LIN {X 0,Y 309.609,Z 476.03,A -85,B 0,C 180,E1 14397.201,E2 14397.201} C_VEL
LIN {X 0,Y 309.614,Z 476.03,A -85,B 0,C 180,E1 14402.807,E2 14402.807} C_VEL
LIN {X 0,Y 308.871,Z 476.03,A -85,B 0,C 180,E1 14411.359,E2 14411.359} C_VEL
LIN {X 0,Y 308.57,Z 476.03,A -85,B 0,C 180,E1 14417.126,E2 14417.126} C_VEL
LIN {X 0,Y 308.226,Z 476.03,A -85,B 0,C 180,E1 14423.143,E2 14423.143} C_VEL
LIN {X 0,Y 307.931,Z 476.03,A -85,B 0,C 180,E1 14429.455,E2 14429.455} C_VEL
LIN {X 0,Y 307.612,Z 476.03,A -85,B 0,C 180,E1 14438.044,E2 14438.044} C_VEL
LIN {X 0,Y 307.589,Z 476.399,A -85,B 0,C 180,E1 14444.592,E2 14444.592} C_VEL
LIN {X 0,Y 310.21,Z 481.903,A -85,B 0,C 180,E1 14445.728,E2 14445.728} C_VEL
LIN {X 0,Y 323.143,Z 502.52,A -85,B 0,C 180,E1 14450.241,E2 14450.241} C_VEL
LIN {X 0,Y 336.192,Z 527.008,A -85,B 0,C 180,E1 14454.493,E2 14454.493} C_VEL
LIN {X 0,Y 347.113,Z 555.503,A -85,B 0,C 180,E1 14458.945,E2 14458.945} C_VEL
LIN {X 0,Y 352.766,Z 578.755,A -85,B 0,C 180,E1 14462.454,E2 14462.454} C_VEL
LIN {X 0,Y 343.722,Z 612.822,A -85,B 0,C 180,E1 14466.127,E2 14466.127} C_VEL
LIN {X 0,Y 334.039,Z 643.34,A -85,B 0,C 180,E1 14470.815,E2 14470.815} C_VEL
LIN {X 0,Y 325.306,Z 668.498,A -85,B 0,C 180,E1 14476.2,E2 14476.2} C_VEL
LIN {X 0,Y 318.194,Z 689.408,A -85,B 0,C 180,E1 14482.481,E2 14482.481} C_VEL
LIN {X 0,Y 313.479,Z 704.958,A -85,B 0,C 180,E1 14489.309,E2 14489.309} C_VEL
LIN {X 0,Y 311.322,Z 714.339,A -85,B 0,C 180,E1 14495.582,E2 14495.582} C_VEL
LIN {X 0,Y 309.931,Z 719.848,A -85,B 0,C 180,E1 14502.293,E2 14502.293} C_VEL
LIN {X 0,Y 309.637,Z 721.106,A -85,B 0,C 180,E1 14507.062,E2 14507.062} C_VEL
LIN {X 0,Y 310.382,Z 718.696,A -85,B 0,C 180,E1 14514.46,E2 14514.46} C_VEL
LIN {X 0,Y 312.319,Z 711.622,A -85,B 0,C 180,E1 14521.411,E2 14521.411} C_VEL
LIN {X 0,Y 316.175,Z 699.192,A -85,B 0,C 180,E1 14528.503,E2 14528.503} C_VEL
LIN {X 0,Y 322.949,Z 681.144,A -85,B 0,C 180,E1 14535.309,E2 14535.309} C_VEL
LIN {X 0,Y 332.145,Z 658.16,A -85,B 0,C 180,E1 14541.336,E2 14541.336} C_VEL
LIN {X 0,Y 342.684,Z 630.258,A -85,B 0,C 180,E1 14546.482,E2 14546.482} C_VEL
LIN {X 0,Y 352.98,Z 599.194,A -85,B 0,C 180,E1 14550.557,E2 14550.557} C_VEL
LIN {X 0,Y 356.508,Z 587.102,A -85,B 0,C 180,E1 14551.803,E2 14551.803} C_VEL
LIN {X 0,Y 356.262,Z 585.186,A -85,B 0,C 180,E1 14552.126,E2 14552.126} C_VEL
LIN {X 0,Y 336.094,Z 594.919,A -85,B 0,C 180,E1 14554.892,E2 14554.892} C_VEL
LIN {X 0,Y 320.136,Z 599.709,A -85,B 0,C 180,E1 14558.13,E2 14558.13} C_VEL
LIN {X 0,Y 319.686,Z 600.582,A -85,B 0,C 180,E1 14558.463,E2 14558.463} C_VEL
LIN {X 0,Y 316.983,Z 624.334,A -85,B 0,C 180,E1 14562.389,E2 14562.389} C_VEL
LIN {X 0,Y 314.808,Z 644.294,A -85,B 0,C 180,E1 14567.144,E2 14567.144} C_VEL
LIN {X 0,Y 313.633,Z 658.734,A -85,B 0,C 180,E1 14572.387,E2 14572.387} C_VEL
LIN {X 0,Y 313.388,Z 666.672,A -85,B 0,C 180,E1 14577.227,E2 14577.227} C_VEL
LIN {X 0,Y 313.677,Z 669.126,A -85,B 0,C 180,E1 14579.996,E2 14579.996} C_VEL
LIN {X 0,Y 314.606,Z 669.657,A -85,B 0,C 180,E1 14585.519,E2 14585.519} C_VEL
LIN {X 0,Y 316.918,Z 664.101,A -85,B 0,C 180,E1 14591.012,E2 14591.012} C_VEL
LIN {X 0,Y 320.125,Z 653.696,A -85,B 0,C 180,E1 14595.776,E2 14595.776} C_VEL
LIN {X 0,Y 324.288,Z 637.409,A -85,B 0,C 180,E1 14600.34,E2 14600.34} C_VEL
LIN {X 0,Y 328.84,Z 615.987,A -85,B 0,C 180,E1 14604.294,E2 14604.294} C_VEL
LIN {X 0,Y 333.119,Z 589.74,A -85,B 0,C 180,E1 14607.559,E2 14607.559} C_VEL
LIN {X 0,Y 336.661,Z 558.53,A -85,B 0,C 180,E1 14610.116,E2 14610.116} C_VEL
LIN {X 0,Y 338.184,Z 535.72,A -85,B 0,C 180,E1 14611.463,E2 14611.463} C_VEL
LIN {X 0,Y 341.71,Z 532.148,A -85,B 0,C 180,E1 14612.114,E2 14612.114} C_VEL
LIN {X 0,Y 344.501,Z 534.122,A -85,B 0,C 180,E1 14613.117,E2 14613.117} C_VEL
LIN {X 0,Y 356.019,Z 559.364,A -85,B 0,C 180,E1 14618.453,E2 14618.453} C_VEL
LIN {X 0,Y 362.184,Z 578.437,A -85,B 0,C 180,E1 14621.558,E2 14621.558} C_VEL
LIN {X 0,Y 351.358,Z 622.491,A -85,B 0,C 180,E1 14624.831,E2 14624.831} C_VEL
LIN {X 0,Y 341.461,Z 657.119,A -85,B 0,C 180,E1 14628.505,E2 14628.505} C_VEL
LIN {X 0,Y 331.204,Z 689.072,A -85,B 0,C 180,E1 14633.283,E2 14633.283} C_VEL
LIN {X 0,Y 322.511,Z 716.02,A -85,B 0,C 180,E1 14638.907,E2 14638.907} C_VEL
LIN {X 0,Y 316.055,Z 737.747,A -85,B 0,C 180,E1 14645.179,E2 14645.179} C_VEL
LIN {X 0,Y 312.202,Z 753.977,A -85,B 0,C 180,E1 14651.794,E2 14651.794} C_VEL
LIN {X 0,Y 310.523,Z 765.226,A -85,B 0,C 180,E1 14658.752,E2 14658.752} C_VEL
LIN {X 0,Y 310.158,Z 770.4,A -85,B 0,C 180,E1 14664.396,E2 14664.396} C_VEL
LIN {X 0,Y 310.336,Z 772.13,A -85,B 0,C 180,E1 14670,E2 14670} C_VEL
LIN {X 0,Y 310.165,Z 770.387,A -85,B 0,C 180,E1 14675.602,E2 14675.602} C_VEL
LIN {X 0,Y 310.766,Z 763.954,A -85,B 0,C 180,E1 14682.17,E2 14682.17} C_VEL
LIN {X 0,Y 312.508,Z 751.967,A -85,B 0,C 180,E1 14688.996,E2 14688.996} C_VEL
LIN {X 0,Y 316.833,Z 733.579,A -85,B 0,C 180,E1 14695.853,E2 14695.853} C_VEL
LIN {X 0,Y 323.626,Z 709.884,A -85,B 0,C 180,E1 14702.054,E2 14702.054} C_VEL
LIN {X 0,Y 325.491,Z 703.783,A -85,B 0,C 180,E1 14703.347,E2 14703.347} C_VEL
LIN {X 0,Y 325.165,Z 692.843,A -85,B 0,C 180,E1 14705.761,E2 14705.761} C_VEL
LIN {X 0,Y 325.168,Z 681.265,A -85,B 0,C 180,E1 14708.078,E2 14708.078} C_VEL
LIN {X 0,Y 334.706,Z 649.033,A -85,B 0,C 180,E1 14712.51,E2 14712.51} C_VEL
LIN {X 0,Y 344.112,Z 612.413,A -85,B 0,C 180,E1 14716.096,E2 14716.096} C_VEL
LIN {X 0,Y 351.392,Z 578.99,A -85,B 0,C 180,E1 14718.568,E2 14718.568} C_VEL
LIN {X 0,Y 336.934,Z 544.114,A -85,B 0,C 180,E1 14723.905,E2 14723.905} C_VEL
LIN {X 0,Y 320.974,Z 511.874,A -85,B 0,C 180,E1 14729.732,E2 14729.732} C_VEL
LIN {X 0,Y 306.924,Z 488.255,A -85,B 0,C 180,E1 14735.215,E2 14735.215} C_VEL
LIN {X 0,Y 302.442,Z 481.461,A -85,B 0,C 180,E1 14737.135,E2 14737.135} C_VEL
LIN {X 0,Y 300.284,Z 476.03,A -85,B 0,C 180,E1 14738.37,E2 14738.37} C_VEL
LIN {X 0,Y 300.741,Z 476.03,A -85,B 0,C 180,E1 14745.426,E2 14745.426} C_VEL
LIN {X 0,Y 301.409,Z 476.03,A -85,B 0,C 180,E1 14754.239,E2 14754.239} C_VEL
LIN {X 0,Y 301.9,Z 476.03,A -85,B 0,C 180,E1 14760.004,E2 14760.004} C_VEL
LIN {X 0,Y 301.407,Z 476.03,A -85,B 0,C 180,E1 14765.77,E2 14765.77} C_VEL
LIN {X 0,Y 300.719,Z 476.03,A -85,B 0,C 180,E1 14774.585,E2 14774.585} C_VEL
LIN {X 0,Y 300.42,Z 476.03,A -85,B 0,C 180,E1 14780.662,E2 14780.662} C_VEL
LIN {X 0,Y 300.101,Z 476.03,A -85,B 0,C 180,E1 14787.009,E2 14787.009} C_VEL
LIN {X 0,Y 299.748,Z 476.03,A -85,B 0,C 180,E1 14793.757,E2 14793.757} C_VEL
LIN {X 0,Y 299.724,Z 476.285,A -85,B 0,C 180,E1 14802.203,E2 14802.203} C_VEL
LIN {X 0,Y 302.277,Z 481.846,A -85,B 0,C 180,E1 14803.462,E2 14803.462} C_VEL
LIN {X 0,Y 316.05,Z 503.587,A -85,B 0,C 180,E1 14808.7,E2 14808.7} C_VEL
LIN {X 0,Y 328.607,Z 526.591,A -85,B 0,C 180,E1 14813.002,E2 14813.002} C_VEL
LIN {X 0,Y 339.745,Z 555.047,A -85,B 0,C 180,E1 14817.67,E2 14817.67} C_VEL
LIN {X 0,Y 346.253,Z 581.175,A -85,B 0,C 180,E1 14821.795,E2 14821.795} C_VEL
LIN {X 0,Y 336.754,Z 615.416,A -85,B 0,C 180,E1 14825.601,E2 14825.601} C_VEL
LIN {X 0,Y 327.378,Z 643.814,A -85,B 0,C 180,E1 14830.057,E2 14830.057} C_VEL
LIN {X 0,Y 318.262,Z 669.058,A -85,B 0,C 180,E1 14835.537,E2 14835.537} C_VEL
LIN {X 0,Y 311.113,Z 689.02,A -85,B 0,C 180,E1 14841.605,E2 14841.605} C_VEL
LIN {X 0,Y 306,Z 704.987,A -85,B 0,C 180,E1 14848.583,E2 14848.583} C_VEL
LIN {X 0,Y 303.42,Z 715.365,A -85,B 0,C 180,E1 14855.728,E2 14855.728} C_VEL
LIN {X 0,Y 302.19,Z 720.102,A -85,B 0,C 180,E1 14861.562,E2 14861.562} C_VEL
LIN {X 0,Y 301.746,Z 721.759,A -85,B 0,C 180,E1 14867.561,E2 14867.561} C_VEL
LIN {X 0,Y 302.329,Z 719.996,A -85,B 0,C 180,E1 14873.62,E2 14873.62} C_VEL
LIN {X 0,Y 303.926,Z 714.692,A -85,B 0,C 180,E1 14879.881,E2 14879.881} C_VEL
LIN {X 0,Y 307.433,Z 703.637,A -85,B 0,C 180,E1 14887.234,E2 14887.234} C_VEL
LIN {X 0,Y 313.533,Z 688.033,A -85,B 0,C 180,E1 14893.962,E2 14893.962} C_VEL
LIN {X 0,Y 322.849,Z 665.785,A -85,B 0,C 180,E1 14900.564,E2 14900.564} C_VEL
LIN {X 0,Y 333.538,Z 639.537,A -85,B 0,C 180,E1 14905.973,E2 14905.973} C_VEL
LIN {X 0,Y 344.606,Z 608.868,A -85,B 0,C 180,E1 14910.476,E2 14910.476} C_VEL
LIN {X 0,Y 349.077,Z 594.477,A -85,B 0,C 180,E1 14912.099,E2 14912.099} C_VEL
LIN {X 0,Y 330.37,Z 602.428,A -85,B 0,C 180,E1 14914.84,E2 14914.84} C_VEL
LIN {X 0,Y 312.096,Z 607.854,A -85,B 0,C 180,E1 14918.66,E2 14918.66} C_VEL
LIN {X 0,Y 311.303,Z 607.869,A -85,B 0,C 180,E1 14919.07,E2 14919.07} C_VEL
LIN {X 0,Y 308.724,Z 630.581,A -85,B 0,C 180,E1 14923.25,E2 14923.25} C_VEL
LIN {X 0,Y 306.627,Z 649.378,A -85,B 0,C 180,E1 14928.244,E2 14928.244} C_VEL
LIN {X 0,Y 305.671,Z 662.626,A -85,B 0,C 180,E1 14933.703,E2 14933.703} C_VEL
LIN {X 0,Y 305.672,Z 669.315,A -85,B 0,C 180,E1 14938.577,E2 14938.577} C_VEL
LIN {X 0,Y 306.155,Z 671.615,A -85,B 0,C 180,E1 14942.83,E2 14942.83} C_VEL
LIN {X 0,Y 308.063,Z 669.42,A -85,B 0,C 180,E1 14948.474,E2 14948.474} C_VEL
LIN {X 0,Y 310.599,Z 662.704,A -85,B 0,C 180,E1 14953.214,E2 14953.214} C_VEL
LIN {X 0,Y 314.735,Z 649.762,A -85,B 0,C 180,E1 14958.216,E2 14958.216} C_VEL
LIN {X 0,Y 319.414,Z 631.57,A -85,B 0,C 180,E1 14962.647,E2 14962.647} C_VEL
LIN {X 0,Y 324.414,Z 607.766,A -85,B 0,C 180,E1 14966.5,E2 14966.5} C_VEL
LIN {X 0,Y 329.026,Z 578.611,A -85,B 0,C 180,E1 14969.642,E2 14969.642} C_VEL
LIN {X 0,Y 332.117,Z 551.912,A -85,B 0,C 180,E1 14971.589,E2 14971.589} C_VEL
LIN {X 0,Y 337.468,Z 544.738,A -85,B 0,C 180,E1 14972.309,E2 14972.309} C_VEL
LIN {X 0,Y 340.537,Z 540.572,A -85,B 0,C 180,E1 14972.717,E2 14972.717} C_VEL
LIN {X 0,Y 351.596,Z 566.201,A -85,B 0,C 180,E1 14978.236,E2 14978.236} C_VEL
LIN {X 0,Y 356.147,Z 581.6,A -85,B 0,C 180,E1 14980.796,E2 14980.796} C_VEL
LIN {X 0,Y 345.155,Z 624.579,A -85,B 0,C 180,E1 14984.082,E2 14984.082} C_VEL
LIN {X 0,Y 334.669,Z 659.139,A -85,B 0,C 180,E1 14987.876,E2 14987.876} C_VEL
LIN {X 0,Y 324.287,Z 689.876,A -85,B 0,C 180,E1 14992.628,E2 14992.628} C_VEL
LIN {X 0,Y 315.042,Z 716.939,A -85,B 0,C 180,E1 14998.486,E2 14998.486} C_VEL
LIN {X 0,Y 308.205,Z 738.6,A -85,B 0,C 180,E1 15005.039,E2 15005.039} C_VEL
LIN {X 0,Y 304.369,Z 754.041,A -85,B 0,C 180,E1 15011.651,E2 15011.651} C_VEL
LIN {X 0,Y 302.674,Z 764.608,A -85,B 0,C 180,E1 15018.457,E2 15018.457} C_VEL
LIN {X 0,Y 302.289,Z 769.775,A -85,B 0,C 180,E1 15024.25,E2 15024.25} C_VEL
LIN {X 0,Y 302.479,Z 771.477,A -85,B 0,C 180,E1 15029.999,E2 15029.999} C_VEL
LIN {X 0,Y 302.296,Z 769.704,A -85,B 0,C 180,E1 15035.749,E2 15035.749} C_VEL
LIN {X 0,Y 302.909,Z 763.208,A -85,B 0,C 180,E1 15042.491,E2 15042.491} C_VEL
LIN {X 0,Y 304.891,Z 750.705,A -85,B 0,C 180,E1 15049.695,E2 15049.695} C_VEL
LIN {X 0,Y 309.48,Z 732.625,A -85,B 0,C 180,E1 15056.515,E2 15056.515} C_VEL
LIN {X 0,Y 316.823,Z 708.164,A -85,B 0,C 180,E1 15062.982,E2 15062.982} C_VEL
LIN {X 0,Y 325.168,Z 681.265,A -85,B 0,C 180,E1 15068.078,E2 15068.078} C_VEL
LIN {X 0,Y 325.431,Z 669.165,A -85,B 0,C 180,E1 15070.295,E2 15070.295} C_VEL
LIN {X 0,Y 325.964,Z 656.299,A -85,B 0,C 180,E1 15072.402,E2 15072.402} C_VEL
LIN {X 0,Y 335.65,Z 620.882,A -85,B 0,C 180,E1 15076.199,E2 15076.199} C_VEL
LIN {X 0,Y 344.722,Z 581.453,A -85,B 0,C 180,E1 15079.278,E2 15079.278} C_VEL
LIN {X 0,Y 330.067,Z 545.357,A -85,B 0,C 180,E1 15085.046,E2 15085.046} C_VEL
LIN {X 0,Y 313.615,Z 512.289,A -85,B 0,C 180,E1 15091.422,E2 15091.422} C_VEL
LIN {X 0,Y 299.519,Z 488.628,A -85,B 0,C 180,E1 15097.433,E2 15097.433} C_VEL
LIN {X 0,Y 295.081,Z 481.89,A -85,B 0,C 180,E1 15099.546,E2 15099.546} C_VEL
LIN {X 0,Y 292.539,Z 476.847,A -85,B 0,C 180,E1 15100.936,E2 15100.936} C_VEL
LIN {X 0,Y 293.021,Z 476.03,A -85,B 0,C 180,E1 15108.077,E2 15108.077} C_VEL
LIN {X 0,Y 293.78,Z 476.03,A -85,B 0,C 180,E1 15117.05,E2 15117.05} C_VEL
LIN {X 0,Y 293.784,Z 476.03,A -85,B 0,C 180,E1 15122.959,E2 15122.959} C_VEL
LIN {X 0,Y 293.006,Z 476.03,A -85,B 0,C 180,E1 15131.933,E2 15131.933} C_VEL
LIN {X 0,Y 292.595,Z 476.03,A -85,B 0,C 180,E1 15138.092,E2 15138.092} C_VEL
LIN {X 0,Y 292.254,Z 476.03,A -85,B 0,C 180,E1 15144.489,E2 15144.489} C_VEL
LIN {X 0,Y 291.907,Z 476.03,A -85,B 0,C 180,E1 15151.248,E2 15151.248} C_VEL
LIN {X 0,Y 291.695,Z 476.599,A -85,B 0,C 180,E1 15159.469,E2 15159.469} C_VEL
LIN {X 0,Y 294.432,Z 481.909,A -85,B 0,C 180,E1 15160.944,E2 15160.944} C_VEL
LIN {X 0,Y 296.791,Z 485.38,A -85,B 0,C 180,E1 15162.033,E2 15162.033} C_VEL
LIN {X 0,Y 311.187,Z 508.02,A -85,B 0,C 180,E1 15167.826,E2 15167.826} C_VEL
LIN {X 0,Y 324.016,Z 532.777,A -85,B 0,C 180,E1 15172.6,E2 15172.6} C_VEL
LIN {X 0,Y 334.089,Z 559.936,A -85,B 0,C 180,E1 15177.227,E2 15177.227} C_VEL
LIN {X 0,Y 339.968,Z 582.863,A -85,B 0,C 180,E1 15181.039,E2 15181.039} C_VEL
LIN {X 0,Y 330.175,Z 616.851,A -85,B 0,C 180,E1 15184.901,E2 15184.901} C_VEL
LIN {X 0,Y 320.145,Z 645.971,A -85,B 0,C 180,E1 15189.587,E2 15189.587} C_VEL
LIN {X 0,Y 310.77,Z 670.877,A -85,B 0,C 180,E1 15195.18,E2 15195.18} C_VEL
LIN {X 0,Y 302.749,Z 692.405,A -85,B 0,C 180,E1 15202.095,E2 15202.095} C_VEL
LIN {X 0,Y 297.782,Z 707.44,A -85,B 0,C 180,E1 15209.272,E2 15209.272} C_VEL
LIN {X 0,Y 295.518,Z 716.37,A -85,B 0,C 180,E1 15215.882,E2 15215.882} C_VEL
LIN {X 0,Y 294.221,Z 721.086,A -85,B 0,C 180,E1 15222.1,E2 15222.1} C_VEL
LIN {X 0,Y 293.861,Z 722.38,A -85,B 0,C 180,E1 15228.009,E2 15228.009} C_VEL
LIN {X 0,Y 294.604,Z 720.448,A -85,B 0,C 180,E1 15234.278,E2 15234.278} C_VEL
LIN {X 0,Y 296.845,Z 713.478,A -85,B 0,C 180,E1 15241.937,E2 15241.937} C_VEL
LIN {X 0,Y 301.07,Z 701.705,A -85,B 0,C 180,E1 15249.215,E2 15249.215} C_VEL
LIN {X 0,Y 308.313,Z 684.584,A -85,B 0,C 180,E1 15256.176,E2 15256.176} C_VEL
LIN {X 0,Y 318.22,Z 662.37,A -85,B 0,C 180,E1 15262.418,E2 15262.418} C_VEL
LIN {X 0,Y 329.501,Z 635.565,A -85,B 0,C 180,E1 15267.723,E2 15267.723} C_VEL
LIN {X 0,Y 340.628,Z 605.233,A -85,B 0,C 180,E1 15271.958,E2 15271.958} C_VEL
LIN {X 0,Y 338.109,Z 604.898,A -85,B 0,C 180,E1 15272.565,E2 15272.565} C_VEL
LIN {X 0,Y 322.886,Z 610.379,A -85,B 0,C 180,E1 15275.034,E2 15275.034} C_VEL
LIN {X 0,Y 303.033,Z 615.082,A -85,B 0,C 180,E1 15279.715,E2 15279.715} C_VEL
LIN {X 0,Y 300.125,Z 638.828,A -85,B 0,C 180,E1 15284.74,E2 15284.74} C_VEL
LIN {X 0,Y 298.442,Z 655.134,A -85,B 0,C 180,E1 15289.768,E2 15289.768} C_VEL
LIN {X 0,Y 297.807,Z 665.902,A -85,B 0,C 180,E1 15294.891,E2 15294.891} C_VEL
LIN {X 0,Y 298.135,Z 671.711,A -85,B 0,C 180,E1 15299.996,E2 15299.996} C_VEL
LIN {X 0,Y 299.258,Z 672.874,A -85,B 0,C 180,E1 15305.803,E2 15305.803} C_VEL
LIN {X 0,Y 301.946,Z 667.982,A -85,B 0,C 180,E1 15311.566,E2 15311.566} C_VEL
LIN {X 0,Y 305.614,Z 658.229,A -85,B 0,C 180,E1 15316.546,E2 15316.546} C_VEL
LIN {X 0,Y 310.068,Z 643.917,A -85,B 0,C 180,E1 15321.018,E2 15321.018} C_VEL
LIN {X 0,Y 315.358,Z 623.654,A -85,B 0,C 180,E1 15325.214,E2 15325.214} C_VEL
LIN {X 0,Y 320.604,Z 598.536,A -85,B 0,C 180,E1 15328.733,E2 15328.733} C_VEL
LIN {X 0,Y 325.036,Z 569.44,A -85,B 0,C 180,E1 15331.5,E2 15331.5} C_VEL
LIN {X 0,Y 332.227,Z 559.13,A -85,B 0,C 180,E1 15332.564,E2 15332.564} C_VEL
LIN {X 0,Y 338.121,Z 551.179,A -85,B 0,C 180,E1 15333.261,E2 15333.261} C_VEL
LIN {X 0,Y 346.556,Z 571.323,A -85,B 0,C 180,E1 15337.702,E2 15337.702} C_VEL
LIN {X 0,Y 350.224,Z 584.949,A -85,B 0,C 180,E1 15340.026,E2 15340.026} C_VEL
LIN {X 0,Y 338.701,Z 627.798,A -85,B 0,C 180,E1 15343.411,E2 15343.411} C_VEL
LIN {X 0,Y 327.65,Z 662.04,A -85,B 0,C 180,E1 15347.337,E2 15347.337} C_VEL
LIN {X 0,Y 316.474,Z 693.235,A -85,B 0,C 180,E1 15352.433,E2 15352.433} C_VEL
LIN {X 0,Y 307.059,Z 719.211,A -85,B 0,C 180,E1 15358.404,E2 15358.404} C_VEL
LIN {X 0,Y 300.103,Z 740.344,A -85,B 0,C 180,E1 15365.232,E2 15365.232} C_VEL
LIN {X 0,Y 296.261,Z 755.274,A -85,B 0,C 180,E1 15372.142,E2 15372.142} C_VEL
LIN {X 0,Y 294.639,Z 765.62,A -85,B 0,C 180,E1 15379.638,E2 15379.638} C_VEL
LIN {X 0,Y 294.403,Z 769.151,A -85,B 0,C 180,E1 15384.096,E2 15384.096} C_VEL
LIN {X 0,Y 294.601,Z 770.82,A -85,B 0,C 180,E1 15389.999,E2 15389.999} C_VEL
LIN {X 0,Y 294.414,Z 769.013,A -85,B 0,C 180,E1 15395.903,E2 15395.903} C_VEL
LIN {X 0,Y 295.046,Z 762.407,A -85,B 0,C 180,E1 15402.867,E2 15402.867} C_VEL
LIN {X 0,Y 297.259,Z 749.623,A -85,B 0,C 180,E1 15410.332,E2 15410.332} C_VEL
LIN {X 0,Y 302.5,Z 730.542,A -85,B 0,C 180,E1 15417.567,E2 15417.567} C_VEL
LIN {X 0,Y 309.973,Z 706.75,A -85,B 0,C 180,E1 15423.875,E2 15423.875} C_VEL
LIN {X 0,Y 319.709,Z 676.68,A -85,B 0,C 180,E1 15429.522,E2 15429.522} C_VEL
LIN {X 0,Y 325.964,Z 656.299,A -85,B 0,C 180,E1 15432.402,E2 15432.402} C_VEL
LIN {X 0,Y 326.557,Z 642.972,A -85,B 0,C 180,E1 15434.403,E2 15434.403} C_VEL
LIN {X 0,Y 326.762,Z 630.968,A -85,B 0,C 180,E1 15436.086,E2 15436.086} C_VEL
LIN {X 0,Y 327.217,Z 629.108,A -85,B 0,C 180,E1 15436.279,E2 15436.279} C_VEL
LIN {X 0,Y 338.217,Z 586.314,A -85,B 0,C 180,E1 15439.759,E2 15439.759} C_VEL
LIN {X 0,Y 330.827,Z 564.854,A -85,B 0,C 180,E1 15443.088,E2 15443.088} C_VEL
LIN {X 0,Y 316.237,Z 532.109,A -85,B 0,C 180,E1 15449.03,E2 15449.03} C_VEL
LIN {X 0,Y 302.744,Z 506.704,A -85,B 0,C 180,E1 15454.763,E2 15454.763} C_VEL
LIN {X 0,Y 291.725,Z 488.604,A -85,B 0,C 180,E1 15460.049,E2 15460.049} C_VEL
LIN {X 0,Y 287.735,Z 482.27,A -85,B 0,C 180,E1 15462.218,E2 15462.218} C_VEL
LIN {X 0,Y 284.853,Z 477.159,A -85,B 0,C 180,E1 15463.996,E2 15463.996} C_VEL
LIN {X 0,Y 284.828,Z 476.03,A -85,B 0,C 180,E1 15464.592,E2 15464.592} C_VEL
LIN {X 0,Y 285.249,Z 476.03,A -85,B 0,C 180,E1 15470.843,E2 15470.843} C_VEL
LIN {X 0,Y 285.872,Z 476.03,A -85,B 0,C 180,E1 15476.969,E2 15476.969} C_VEL
LIN {X 0,Y 285.876,Z 476.03,A -85,B 0,C 180,E1 15483.04,E2 15483.04} C_VEL
LIN {X 0,Y 285.039,Z 476.03,A -85,B 0,C 180,E1 15492.272,E2 15492.272} C_VEL
LIN {X 0,Y 284.633,Z 476.03,A -85,B 0,C 180,E1 15498.616,E2 15498.616} C_VEL
LIN {X 0,Y 284.224,Z 476.03,A -85,B 0,C 180,E1 15505.228,E2 15505.228} C_VEL
LIN {X 0,Y 283.914,Z 476.03,A -85,B 0,C 180,E1 15512.232,E2 15512.232} C_VEL
LIN {X 0,Y 283.745,Z 476.662,A -85,B 0,C 180,E1 15516.321,E2 15516.321} C_VEL
LIN {X 0,Y 286.301,Z 481.851,A -85,B 0,C 180,E1 15517.935,E2 15517.935} C_VEL
LIN {X 0,Y 288.695,Z 484.966,A -85,B 0,C 180,E1 15519.171,E2 15519.171} C_VEL
LIN {X 0,Y 296.918,Z 497.495,A -85,B 0,C 180,E1 15523.117,E2 15523.117} C_VEL
LIN {X 0,Y 311.191,Z 521.574,A -85,B 0,C 180,E1 15528.821,E2 15528.821} C_VEL
LIN {X 0,Y 322.531,Z 546.631,A -85,B 0,C 180,E1 15533.62,E2 15533.62} C_VEL
LIN {X 0,Y 331.022,Z 574.59,A -85,B 0,C 180,E1 15538.464,E2 15538.464} C_VEL
LIN {X 0,Y 333.111,Z 586.916,A -85,B 0,C 180,E1 15540.488,E2 15540.488} C_VEL
LIN {X 0,Y 322.86,Z 620.465,A -85,B 0,C 180,E1 15544.478,E2 15544.478} C_VEL
LIN {X 0,Y 312.305,Z 649.755,A -85,B 0,C 180,E1 15549.422,E2 15549.422} C_VEL
LIN {X 0,Y 302.309,Z 675.137,A -85,B 0,C 180,E1 15555.498,E2 15555.498} C_VEL
LIN {X 0,Y 295.014,Z 693.864,A -85,B 0,C 180,E1 15561.887,E2 15561.887} C_VEL
LIN {X 0,Y 289.935,Z 708.672,A -85,B 0,C 180,E1 15569.252,E2 15569.252} C_VEL
LIN {X 0,Y 287.606,Z 717.372,A -85,B 0,C 180,E1 15576.044,E2 15576.044} C_VEL
LIN {X 0,Y 286.332,Z 721.818,A -85,B 0,C 180,E1 15582.212,E2 15582.212} C_VEL
LIN {X 0,Y 285.97,Z 723.003,A -85,B 0,C 180,E1 15588.523,E2 15588.523} C_VEL
LIN {X 0,Y 287.228,Z 719.947,A -85,B 0,C 180,E1 15596.341,E2 15596.341} C_VEL
LIN {X 0,Y 289.963,Z 712.048,A -85,B 0,C 180,E1 15604.014,E2 15604.014} C_VEL
LIN {X 0,Y 295.487,Z 698.518,A -85,B 0,C 180,E1 15611.77,E2 15611.77} C_VEL
LIN {X 0,Y 304.141,Z 679.702,A -85,B 0,C 180,E1 15618.818,E2 15618.818} C_VEL
LIN {X 0,Y 314.888,Z 656.582,A -85,B 0,C 180,E1 15624.83,E2 15624.83} C_VEL
LIN {X 0,Y 327.425,Z 627.238,A -85,B 0,C 180,E1 15630.138,E2 15630.138} C_VEL
LIN {X 0,Y 332.667,Z 613.469,A -85,B 0,C 180,E1 15632.053,E2 15632.053} C_VEL
LIN {X 0,Y 322.212,Z 615.964,A -85,B 0,C 180,E1 15633.958,E2 15633.958} C_VEL
LIN {X 0,Y 298.724,Z 621.958,A -85,B 0,C 180,E1 15639.215,E2 15639.215} C_VEL
LIN {X 0,Y 294.437,Z 622.432,A -85,B 0,C 180,E1 15640.665,E2 15640.665} C_VEL
LIN {X 0,Y 291.833,Z 644.216,A -85,B 0,C 180,E1 15645.729,E2 15645.729} C_VEL
LIN {X 0,Y 290.368,Z 659.482,A -85,B 0,C 180,E1 15650.996,E2 15650.996} C_VEL
LIN {X 0,Y 289.999,Z 670.065,A -85,B 0,C 180,E1 15657.003,E2 15657.003} C_VEL
LIN {X 0,Y 290.37,Z 672.995,A -85,B 0,C 180,E1 15659.995,E2 15659.995} C_VEL
LIN {X 0,Y 291.585,Z 674.478,A -85,B 0,C 180,E1 15665.956,E2 15665.956} C_VEL
LIN {X 0,Y 294.451,Z 669.947,A -85,B 0,C 180,E1 15671.864,E2 15671.864} C_VEL
LIN {X 0,Y 298.408,Z 660.544,A -85,B 0,C 180,E1 15676.957,E2 15676.957} C_VEL
LIN {X 0,Y 303.782,Z 644.865,A -85,B 0,C 180,E1 15682.007,E2 15682.007} C_VEL
LIN {X 0,Y 309.846,Z 623.218,A -85,B 0,C 180,E1 15686.475,E2 15686.475} C_VEL
LIN {X 0,Y 315.564,Z 597.737,A -85,B 0,C 180,E1 15690.005,E2 15690.005} C_VEL
LIN {X 0,Y 318.84,Z 581.686,A -85,B 0,C 180,E1 15691.703,E2 15691.703} C_VEL
LIN {X 0,Y 325.435,Z 574.296,A -85,B 0,C 180,E1 15692.636,E2 15692.636} C_VEL
LIN {X 0,Y 335.517,Z 561.337,A -85,B 0,C 180,E1 15693.782,E2 15693.782} C_VEL
LIN {X 0,Y 343.109,Z 581.621,A -85,B 0,C 180,E1 15698.148,E2 15698.148} C_VEL
LIN {X 0,Y 344.6,Z 587.31,A -85,B 0,C 180,E1 15699.158,E2 15699.158} C_VEL
LIN {X 0,Y 332.771,Z 629.408,A -85,B 0,C 180,E1 15702.562,E2 15702.562} C_VEL
LIN {X 0,Y 321.142,Z 663.568,A -85,B 0,C 180,E1 15706.594,E2 15706.594} C_VEL
LIN {X 0,Y 309.424,Z 694.498,A -85,B 0,C 180,E1 15711.822,E2 15711.822} C_VEL
LIN {X 0,Y 299.602,Z 720.094,A -85,B 0,C 180,E1 15717.95,E2 15717.95} C_VEL
LIN {X 0,Y 292.308,Z 740.975,A -85,B 0,C 180,E1 15725.023,E2 15725.023} C_VEL
LIN {X 0,Y 288.248,Z 755.995,A -85,B 0,C 180,E1 15732.419,E2 15732.419} C_VEL
LIN {X 0,Y 286.796,Z 765.011,A -85,B 0,C 180,E1 15739.351,E2 15739.351} C_VEL
LIN {X 0,Y 286.536,Z 768.535,A -85,B 0,C 180,E1 15743.933,E2 15743.933} C_VEL
LIN {X 0,Y 286.742,Z 770.165,A -85,B 0,C 180,E1 15749.999,E2 15749.999} C_VEL
LIN {X 0,Y 286.545,Z 768.322,A -85,B 0,C 180,E1 15756.066,E2 15756.066} C_VEL
LIN {X 0,Y 287.186,Z 761.639,A -85,B 0,C 180,E1 15763.226,E2 15763.226} C_VEL
LIN {X 0,Y 289.614,Z 748.777,A -85,B 0,C 180,E1 15770.887,E2 15770.887} C_VEL
LIN {X 0,Y 295.027,Z 730.055,A -85,B 0,C 180,E1 15778.141,E2 15778.141} C_VEL
LIN {X 0,Y 303.169,Z 705.604,A -85,B 0,C 180,E1 15784.743,E2 15784.743} C_VEL
LIN {X 0,Y 312.99,Z 676.292,A -85,B 0,C 180,E1 15790.317,E2 15790.317} C_VEL
LIN {X 0,Y 323.394,Z 642.954,A -85,B 0,C 180,E1 15794.821,E2 15794.821} C_VEL
LIN {X 0,Y 327.217,Z 629.108,A -85,B 0,C 180,E1 15796.279,E2 15796.279} C_VEL
LIN {X 0,Y 328.139,Z 614.723,A -85,B 0,C 180,E1 15798.031,E2 15798.031} C_VEL
LIN {X 0,Y 328.953,Z 599.932,A -85,B 0,C 180,E1 15799.669,E2 15799.669} C_VEL
LIN {X 0,Y 331.587,Z 586.783,A -85,B 0,C 180,E1 15800.728,E2 15800.728} C_VEL
LIN {X 0,Y 317.907,Z 551.766,A -85,B 0,C 180,E1 15806.797,E2 15806.797} C_VEL
LIN {X 0,Y 303.981,Z 522.544,A -85,B 0,C 180,E1 15812.891,E2 15812.891} C_VEL
LIN {X 0,Y 291.587,Z 500.707,A -85,B 0,C 180,E1 15818.831,E2 15818.831} C_VEL
LIN {X 0,Y 284.057,Z 488.673,A -85,B 0,C 180,E1 15822.976,E2 15822.976} C_VEL
LIN {X 0,Y 280.379,Z 482.542,A -85,B 0,C 180,E1 15825.343,E2 15825.343} C_VEL
LIN {X 0,Y 277.277,Z 477.708,A -85,B 0,C 180,E1 15827.472,E2 15827.472} C_VEL
LIN {X 0,Y 277.136,Z 476.03,A -85,B 0,C 180,E1 15828.045,E2 15828.045} C_VEL
LIN {X 0,Y 277.943,Z 476.03,A -85,B 0,C 180,E1 15836.882,E2 15836.882} C_VEL
LIN {X 0,Y 277.947,Z 476.03,A -85,B 0,C 180,E1 15843.127,E2 15843.127} C_VEL
LIN {X 0,Y 277.073,Z 476.03,A -85,B 0,C 180,E1 15852.63,E2 15852.63} C_VEL
LIN {X 0,Y 276.497,Z 476.03,A -85,B 0,C 180,E1 15861.421,E2 15861.421} C_VEL
LIN {X 0,Y 276.082,Z 476.03,A -85,B 0,C 180,E1 15869.58,E2 15869.58} C_VEL
LIN {X 0,Y 275.958,Z 476.521,A -85,B 0,C 180,E1 15872.571,E2 15872.571} C_VEL
LIN {X 0,Y 278.26,Z 481.759,A -85,B 0,C 180,E1 15874.42,E2 15874.42} C_VEL
LIN {X 0,Y 280.861,Z 484.837,A -85,B 0,C 180,E1 15875.982,E2 15875.982} C_VEL
LIN {X 0,Y 289.685,Z 498.023,A -85,B 0,C 180,E1 15880.804,E2 15880.804} C_VEL
LIN {X 0,Y 304.465,Z 522.84,A -85,B 0,C 180,E1 15887.274,E2 15887.274} C_VEL
LIN {X 0,Y 315.256,Z 546.247,A -85,B 0,C 180,E1 15892.058,E2 15892.058} C_VEL
LIN {X 0,Y 323.782,Z 573.558,A -85,B 0,C 180,E1 15897.036,E2 15897.036} C_VEL
LIN {X 0,Y 326.953,Z 588.092,A -85,B 0,C 180,E1 15899.626,E2 15899.626} C_VEL
LIN {X 0,Y 316.727,Z 620.742,A -85,B 0,C 180,E1 15903.565,E2 15903.565} C_VEL
LIN {X 0,Y 306.396,Z 648.51,A -85,B 0,C 180,E1 15908.246,E2 15908.246} C_VEL
LIN {X 0,Y 295.828,Z 674.469,A -85,B 0,C 180,E1 15914.413,E2 15914.413} C_VEL
LIN {X 0,Y 287.998,Z 693.581,A -85,B 0,C 180,E1 15920.926,E2 15920.926} C_VEL
LIN {X 0,Y 282.436,Z 708.678,A -85,B 0,C 180,E1 15928.465,E2 15928.465} C_VEL
LIN {X 0,Y 279.697,Z 718.368,A -85,B 0,C 180,E1 15936.216,E2 15936.216} C_VEL
LIN {X 0,Y 278.399,Z 722.653,A -85,B 0,C 180,E1 15942.566,E2 15942.566} C_VEL
LIN {X 0,Y 278.107,Z 723.626,A -85,B 0,C 180,E1 15949.067,E2 15949.067} C_VEL
LIN {X 0,Y 279.557,Z 720.331,A -85,B 0,C 180,E1 15957.123,E2 15957.123} C_VEL
LIN {X 0,Y 282.716,Z 712.051,A -85,B 0,C 180,E1 15965.102,E2 15965.102} C_VEL
LIN {X 0,Y 288.827,Z 698.228,A -85,B 0,C 180,E1 15972.962,E2 15972.962} C_VEL
LIN {X 0,Y 298.233,Z 679.074,A -85,B 0,C 180,E1 15980.133,E2 15980.133} C_VEL
LIN {X 0,Y 310.22,Z 654.487,A -85,B 0,C 180,E1 15986.424,E2 15986.424} C_VEL
LIN {X 0,Y 322.479,Z 626.679,A -85,B 0,C 180,E1 15991.353,E2 15991.353} C_VEL
LIN {X 0,Y 324.961,Z 620.358,A -85,B 0,C 180,E1 15992.287,E2 15992.287} C_VEL
LIN {X 0,Y 297.852,Z 627.4,A -85,B 0,C 180,E1 15997.834,E2 15997.834} C_VEL
LIN {X 0,Y 285.93,Z 629.711,A -85,B 0,C 180,E1 16001.697,E2 16001.697} C_VEL
LIN {X 0,Y 283.539,Z 649.617,A -85,B 0,C 180,E1 16006.878,E2 16006.878} C_VEL
LIN {X 0,Y 282.404,Z 663.433,A -85,B 0,C 180,E1 16012.238,E2 16012.238} C_VEL
LIN {X 0,Y 282.192,Z 671.157,A -85,B 0,C 180,E1 16016.92,E2 16016.92} C_VEL
LIN {X 0,Y 282.571,Z 674.259,A -85,B 0,C 180,E1 16019.995,E2 16019.995} C_VEL
LIN {X 0,Y 283.906,Z 676.095,A -85,B 0,C 180,E1 16026.118,E2 16026.118} C_VEL
LIN {X 0,Y 286.981,Z 671.927,A -85,B 0,C 180,E1 16032.178,E2 16032.178} C_VEL
LIN {X 0,Y 291.212,Z 662.922,A -85,B 0,C 180,E1 16037.389,E2 16037.389} C_VEL
LIN {X 0,Y 296.884,Z 648.017,A -85,B 0,C 180,E1 16042.482,E2 16042.482} C_VEL
LIN {X 0,Y 303.474,Z 627.02,A -85,B 0,C 180,E1 16047.075,E2 16047.075} C_VEL
LIN {X 0,Y 310.112,Z 600.787,A -85,B 0,C 180,E1 16050.9,E2 16050.9} C_VEL
LIN {X 0,Y 311.364,Z 595.307,A -85,B 0,C 180,E1 16051.543,E2 16051.543} C_VEL
LIN {X 0,Y 317.528,Z 589.368,A -85,B 0,C 180,E1 16052.537,E2 16052.537} C_VEL
LIN {X 0,Y 333.101,Z 571.806,A -85,B 0,C 180,E1 16054.483,E2 16054.483} C_VEL
LIN {X 0,Y 338.742,Z 589.606,A -85,B 0,C 180,E1 16058.191,E2 16058.191} C_VEL
LIN {X 0,Y 326.93,Z 631.065,A -85,B 0,C 180,E1 16061.685,E2 16061.685} C_VEL
LIN {X 0,Y 314.461,Z 665.679,A -85,B 0,C 180,E1 16065.901,E2 16065.901} C_VEL
LIN {X 0,Y 302.143,Z 696.414,A -85,B 0,C 180,E1 16071.324,E2 16071.324} C_VEL
LIN {X 0,Y 291.666,Z 722.249,A -85,B 0,C 180,E1 16077.852,E2 16077.852} C_VEL
LIN {X 0,Y 284.534,Z 741.623,A -85,B 0,C 180,E1 16084.804,E2 16084.804} C_VEL
LIN {X 0,Y 280.256,Z 756.666,A -85,B 0,C 180,E1 16092.713,E2 16092.713} C_VEL
LIN {X 0,Y 278.741,Z 765.787,A -85,B 0,C 180,E1 16100.621,E2 16100.621} C_VEL
LIN {X 0,Y 278.619,Z 769.117,A -85,B 0,C 180,E1 16106.884,E2 16106.884} C_VEL
LIN {X 0,Y 278.675,Z 769.027,A -85,B 0,C 180,E1 16113.114,E2 16113.114} C_VEL
LIN {X 0,Y 278.774,Z 765.351,A -85,B 0,C 180,E1 16119.377,E2 16119.377} C_VEL
LIN {X 0,Y 279.997,Z 756.834,A -85,B 0,C 180,E1 16126.493,E2 16126.493} C_VEL
LIN {X 0,Y 283.899,Z 741.314,A -85,B 0,C 180,E1 16134.414,E2 16134.414} C_VEL
LIN {X 0,Y 290.444,Z 720.953,A -85,B 0,C 180,E1 16141.42,E2 16141.42} C_VEL
LIN {X 0,Y 299.976,Z 694.051,A -85,B 0,C 180,E1 16147.875,E2 16147.875} C_VEL
LIN {X 0,Y 310.542,Z 663.494,A -85,B 0,C 180,E1 16153.047,E2 16153.047} C_VEL
LIN {X 0,Y 321.295,Z 627.983,A -85,B 0,C 180,E1 16157.258,E2 16157.258} C_VEL
LIN {X 0,Y 328.953,Z 599.932,A -85,B 0,C 180,E1 16159.669,E2 16159.669} C_VEL
LIN {X 0,Y 328.313,Z 593.056,A -85,B 0,C 180,E1 16160.563,E2 16160.563} C_VEL
LIN {X 0,Y 322.947,Z 583.585,A -85,B 0,C 180,E1 16162.495,E2 16162.495} C_VEL
LIN {X 0,Y 309.71,Z 549.893,A -85,B 0,C 180,E1 16168.713,E2 16168.713} C_VEL
LIN {X 0,Y 296.538,Z 522.688,A -85,B 0,C 180,E1 16174.892,E2 16174.892} C_VEL
LIN {X 0,Y 285.13,Z 502.326,A -85,B 0,C 180,E1 16180.925,E2 16180.925} C_VEL
LIN {X 0,Y 277.113,Z 489.399,A -85,B 0,C 180,E1 16185.974,E2 16185.974} C_VEL
LIN {X 0,Y 272.941,Z 482.722,A -85,B 0,C 180,E1 16189.085,E2 16189.085} C_VEL
LIN {X 0,Y 269.559,Z 477.497,A -85,B 0,C 180,E1 16192.035,E2 16192.035} C_VEL
LIN {X 0,Y 269.507,Z 476.03,A -85,B 0,C 180,E1 16192.743,E2 16192.743} C_VEL
LIN {X 0,Y 270.327,Z 476.03,A -85,B 0,C 180,E1 16200.005,E2 16200.005} C_VEL
LIN {X 0,Y 269.658,Z 476.03,A -85,B 0,C 180,E1 16206.452,E2 16206.452} C_VEL
LIN {X 0,Y 269.098,Z 476.03,A -85,B 0,C 180,E1 16213.011,E2 16213.011} C_VEL
LIN {X 0,Y 268.654,Z 476.03,A -85,B 0,C 180,E1 16219.768,E2 16219.768} C_VEL
LIN {X 0,Y 268.258,Z 476.56,A -85,B 0,C 180,E1 16227.91,E2 16227.91} C_VEL
LIN {X 0,Y 270.942,Z 482.036,A -85,B 0,C 180,E1 16230.548,E2 16230.548} C_VEL
LIN {X 0,Y 273.149,Z 484.585,A -85,B 0,C 180,E1 16232.192,E2 16232.192} C_VEL
LIN {X 0,Y 276.998,Z 490.129,A -85,B 0,C 180,E1 16234.881,E2 16234.881} C_VEL
LIN {X 0,Y 289.334,Z 509.525,A -85,B 0,C 180,E1 16241.78,E2 16241.78} C_VEL
LIN {X 0,Y 302.879,Z 534.115,A -85,B 0,C 180,E1 16247.904,E2 16247.904} C_VEL
LIN {X 0,Y 312.272,Z 557.606,A -85,B 0,C 180,E1 16252.708,E2 16252.708} C_VEL
LIN {X 0,Y 319.086,Z 583.642,A -85,B 0,C 180,E1 16257.575,E2 16257.575} C_VEL
LIN {X 0,Y 320.066,Z 592.416,A -85,B 0,C 180,E1 16259.094,E2 16259.094} C_VEL
LIN {X 0,Y 309.464,Z 624.283,A -85,B 0,C 180,E1 16263.092,E2 16263.092} C_VEL
LIN {X 0,Y 297.903,Z 653.882,A -85,B 0,C 180,E1 16268.378,E2 16268.378} C_VEL
LIN {X 0,Y 287.316,Z 678.526,A -85,B 0,C 180,E1 16274.723,E2 16274.723} C_VEL
LIN {X 0,Y 279.554,Z 696.756,A -85,B 0,C 180,E1 16281.435,E2 16281.435} C_VEL
LIN {X 0,Y 274.224,Z 711.098,A -85,B 0,C 180,E1 16289.21,E2 16289.21} C_VEL
LIN {X 0,Y 271.778,Z 719.359,A -85,B 0,C 180,E1 16296.398,E2 16296.398} C_VEL
LIN {X 0,Y 270.439,Z 723.43,A -85,B 0,C 180,E1 16302.942,E2 16302.942} C_VEL
LIN {X 0,Y 270.24,Z 724.254,A -85,B 0,C 180,E1 16309.644,E2 16309.644} C_VEL
LIN {X 0,Y 271.646,Z 721.402,A -85,B 0,C 180,E1 16316.895,E2 16316.895} C_VEL
LIN {X 0,Y 274.32,Z 714.754,A -85,B 0,C 180,E1 16324.111,E2 16324.111} C_VEL
LIN {X 0,Y 280.181,Z 702.043,A -85,B 0,C 180,E1 16332.24,E2 16332.24} C_VEL
LIN {X 0,Y 289.851,Z 683.453,A -85,B 0,C 180,E1 16339.903,E2 16339.903} C_VEL
LIN {X 0,Y 301.9,Z 660.141,A -85,B 0,C 180,E1 16346.349,E2 16346.349} C_VEL
LIN {X 0,Y 315.32,Z 631.756,A -85,B 0,C 180,E1 16351.767,E2 16351.767} C_VEL
LIN {X 0,Y 316.514,Z 628.94,A -85,B 0,C 180,E1 16352.196,E2 16352.196} C_VEL
LIN {X 0,Y 314.56,Z 628.495,A -85,B 0,C 180,E1 16352.786,E2 16352.786} C_VEL
LIN {X 0,Y 289.191,Z 634.408,A -85,B 0,C 180,E1 16358.497,E2 16358.497} C_VEL
LIN {X 0,Y 277.501,Z 636.441,A -85,B 0,C 180,E1 16362.776,E2 16362.776} C_VEL
LIN {X 0,Y 275.301,Z 654.646,A -85,B 0,C 180,E1 16368.094,E2 16368.094} C_VEL
LIN {X 0,Y 274.397,Z 667.34,A -85,B 0,C 180,E1 16373.66,E2 16373.66} C_VEL
LIN {X 0,Y 274.779,Z 675.519,A -85,B 0,C 180,E1 16379.995,E2 16379.995} C_VEL
LIN {X 0,Y 276.239,Z 677.722,A -85,B 0,C 180,E1 16386.288,E2 16386.288} C_VEL
LIN {X 0,Y 279.52,Z 673.95,A -85,B 0,C 180,E1 16392.508,E2 16392.508} C_VEL
LIN {X 0,Y 284.066,Z 665.389,A -85,B 0,C 180,E1 16397.841,E2 16397.841} C_VEL
LIN {X 0,Y 290.214,Z 650.777,A -85,B 0,C 180,E1 16403.11,E2 16403.11} C_VEL
LIN {X 0,Y 297.197,Z 631.002,A -85,B 0,C 180,E1 16407.696,E2 16407.696} C_VEL
LIN {X 0,Y 304.219,Z 607.547,A -85,B 0,C 180,E1 16411.424,E2 16411.424} C_VEL
LIN {X 0,Y 319.004,Z 593.784,A -85,B 0,C 180,E1 16413.685,E2 16413.685} C_VEL
LIN {X 0,Y 330.125,Z 582.414,A -85,B 0,C 180,E1 16415.124,E2 16415.124} C_VEL
LIN {X 0,Y 332.943,Z 594.686,A -85,B 0,C 180,E1 16417.521,E2 16417.521} C_VEL
LIN {X 0,Y 320.667,Z 634.201,A -85,B 0,C 180,E1 16420.932,E2 16420.932} C_VEL
LIN {X 0,Y 308.074,Z 667.229,A -85,B 0,C 180,E1 16425.103,E2 16425.103} C_VEL
LIN {X 0,Y 295.469,Z 696.95,A -85,B 0,C 180,E1 16430.5,E2 16430.5} C_VEL
LIN {X 0,Y 284.741,Z 721.856,A -85,B 0,C 180,E1 16436.972,E2 16436.972} C_VEL
LIN {X 0,Y 277.097,Z 741.134,A -85,B 0,C 180,E1 16444.078,E2 16444.078} C_VEL
LIN {X 0,Y 272.513,Z 756.108,A -85,B 0,C 180,E1 16452.206,E2 16452.206} C_VEL
LIN {X 0,Y 270.892,Z 765.18,A -85,B 0,C 180,E1 16460.346,E2 16460.346} C_VEL
LIN {X 0,Y 270.729,Z 768.483,A -85,B 0,C 180,E1 16466.793,E2 16466.793} C_VEL
LIN {X 0,Y 270.81,Z 768.348,A -85,B 0,C 180,E1 16473.205,E2 16473.205} C_VEL
LIN {X 0,Y 270.924,Z 764.616,A -85,B 0,C 180,E1 16479.651,E2 16479.651} C_VEL
LIN {X 0,Y 272.219,Z 756.011,A -85,B 0,C 180,E1 16486.978,E2 16486.978} C_VEL
LIN {X 0,Y 276.395,Z 740.496,A -85,B 0,C 180,E1 16495.069,E2 16495.069} C_VEL
LIN {X 0,Y 283.408,Z 719.865,A -85,B 0,C 180,E1 16502.293,E2 16502.293} C_VEL
LIN {X 0,Y 293.188,Z 693.536,A -85,B 0,C 180,E1 16508.713,E2 16508.713} C_VEL
LIN {X 0,Y 303.902,Z 663.774,A -85,B 0,C 180,E1 16513.844,E2 16513.844} C_VEL
LIN {X 0,Y 314.716,Z 629.564,A -85,B 0,C 180,E1 16518.011,E2 16518.011} C_VEL
LIN {X 0,Y 325.083,Z 589.557,A -85,B 0,C 180,E1 16521.47,E2 16521.47} C_VEL
LIN {X 0,Y 322.947,Z 583.585,A -85,B 0,C 180,E1 16522.495,E2 16522.495} C_VEL
LIN {X 0,Y 317.926,Z 576.204,A -85,B 0,C 180,E1 16524.217,E2 16524.217} C_VEL
LIN {X 0,Y 309.325,Z 566.485,A -85,B 0,C 180,E1 16526.972,E2 16526.972} C_VEL
LIN {X 0,Y 308.707,Z 565.06,A -85,B 0,C 180,E1 16527.262,E2 16527.262} C_VEL
LIN {X 0,Y 295.574,Z 535.091,A -85,B 0,C 180,E1 16533.787,E2 16533.787} C_VEL
LIN {X 0,Y 283.957,Z 513.206,A -85,B 0,C 180,E1 16540.033,E2 16540.033} C_VEL
LIN {X 0,Y 274.43,Z 496.717,A -85,B 0,C 180,E1 16546.241,E2 16546.241} C_VEL
LIN {X 0,Y 269.92,Z 489.701,A -85,B 0,C 180,E1 16549.706,E2 16549.706} C_VEL
LIN {X 0,Y 266.695,Z 483.723,A -85,B 0,C 180,E1 16552.871,E2 16552.871} C_VEL
LIN {X 0,Y 262.361,Z 477.907,A -85,B 0,C 180,E1 16557.731,E2 16557.731} C_VEL
LIN {X 0,Y 262.219,Z 476.03,A -85,B 0,C 180,E1 16558.764,E2 16558.764} C_VEL
LIN {X 0,Y 261.71,Z 476.03,A -85,B 0,C 180,E1 16566.649,E2 16566.649} C_VEL
LIN {X 0,Y 261.131,Z 476.03,A -85,B 0,C 180,E1 16573.415,E2 16573.415} C_VEL
LIN {X 0,Y 260.594,Z 476.798,A -85,B 0,C 180,E1 16581.092,E2 16581.092} C_VEL
LIN {X 0,Y 263.775,Z 482.505,A -85,B 0,C 180,E1 16585.635,E2 16585.635} C_VEL
LIN {X 0,Y 265.831,Z 484.76,A -85,B 0,C 180,E1 16587.686,E2 16587.686} C_VEL
LIN {X 0,Y 269.766,Z 490.363,A -85,B 0,C 180,E1 16591.163,E2 16591.163} C_VEL
LIN {X 0,Y 273.998,Z 497.128,A -85,B 0,C 180,E1 16594.346,E2 16594.346} C_VEL
LIN {X 0,Y 285.811,Z 516.088,A -85,B 0,C 180,E1 16601.226,E2 16601.226} C_VEL
LIN {X 0,Y 298.107,Z 539.326,A -85,B 0,C 180,E1 16607.201,E2 16607.201} C_VEL
LIN {X 0,Y 307.341,Z 563.961,A -85,B 0,C 180,E1 16612.424,E2 16612.424} C_VEL
LIN {X 0,Y 313.871,Z 592.445,A -85,B 0,C 180,E1 16617.952,E2 16617.952} C_VEL
LIN {X 0,Y 306.359,Z 616.68,A -85,B 0,C 180,E1 16620.991,E2 16620.991} C_VEL
LIN {X 0,Y 295.012,Z 645.91,A -85,B 0,C 180,E1 16625.759,E2 16625.759} C_VEL
LIN {X 0,Y 283.755,Z 671.57,A -85,B 0,C 180,E1 16631.731,E2 16631.731} C_VEL
LIN {X 0,Y 274.214,Z 692.796,A -85,B 0,C 180,E1 16638.858,E2 16638.858} C_VEL
LIN {X 0,Y 267.618,Z 708.677,A -85,B 0,C 180,E1 16646.757,E2 16646.757} C_VEL
LIN {X 0,Y 264.261,Z 718.903,A -85,B 0,C 180,E1 16654.931,E2 16654.931} C_VEL
LIN {X 0,Y 262.715,Z 723.49,A -85,B 0,C 180,E1 16661.54,E2 16661.54} C_VEL
LIN {X 0,Y 262.401,Z 724.883,A -85,B 0,C 180,E1 16670.257,E2 16670.257} C_VEL
LIN {X 0,Y 264.394,Z 720.832,A -85,B 0,C 180,E1 16679.129,E2 16679.129} C_VEL
LIN {X 0,Y 268.733,Z 711.278,A -85,B 0,C 180,E1 16687.924,E2 16687.924} C_VEL
LIN {X 0,Y 276.487,Z 696.567,A -85,B 0,C 180,E1 16696.051,E2 16696.051} C_VEL
LIN {X 0,Y 287.872,Z 676.032,A -85,B 0,C 180,E1 16703.443,E2 16703.443} C_VEL
LIN {X 0,Y 300.751,Z 651.778,A -85,B 0,C 180,E1 16709.396,E2 16709.396} C_VEL
LIN {X 0,Y 308.132,Z 636.601,A -85,B 0,C 180,E1 16712.191,E2 16712.191} C_VEL
LIN {X 0,Y 307.694,Z 635.313,A -85,B 0,C 180,E1 16712.679,E2 16712.679} C_VEL
LIN {X 0,Y 284.257,Z 640.449,A -85,B 0,C 180,E1 16718.105,E2 16718.105} C_VEL
LIN {X 0,Y 269.069,Z 642.454,A -85,B 0,C 180,E1 16723.864,E2 16723.864} C_VEL
LIN {X 0,Y 267.164,Z 659.365,A -85,B 0,C 180,E1 16729.382,E2 16729.382} C_VEL
LIN {X 0,Y 266.556,Z 671.135,A -85,B 0,C 180,E1 16735.275,E2 16735.275} C_VEL
LIN {X 0,Y 267.128,Z 677.968,A -85,B 0,C 180,E1 16741.619,E2 16741.619} C_VEL
LIN {X 0,Y 268.568,Z 679.352,A -85,B 0,C 180,E1 16746.469,E2 16746.469} C_VEL
LIN {X 0,Y 272.088,Z 675.991,A -85,B 0,C 180,E1 16752.855,E2 16752.855} C_VEL
LIN {X 0,Y 276.942,Z 667.89,A -85,B 0,C 180,E1 16758.316,E2 16758.316} C_VEL
LIN {X 0,Y 283.949,Z 652.931,A -85,B 0,C 180,E1 16763.984,E2 16763.984} C_VEL
LIN {X 0,Y 291.623,Z 633.287,A -85,B 0,C 180,E1 16768.695,E2 16768.695} C_VEL
LIN {X 0,Y 296.616,Z 618.877,A -85,B 0,C 180,E1 16771.23,E2 16771.23} C_VEL
LIN {X 0,Y 315.197,Z 603.587,A -85,B 0,C 180,E1 16774.193,E2 16774.193} C_VEL
LIN {X 0,Y 325.89,Z 592.946,A -85,B 0,C 180,E1 16775.496,E2 16775.496} C_VEL
LIN {X 0,Y 327.578,Z 596.691,A -85,B 0,C 180,E1 16776.512,E2 16776.512} C_VEL
LIN {X 0,Y 315.489,Z 634.423,A -85,B 0,C 180,E1 16779.835,E2 16779.835} C_VEL
LIN {X 0,Y 302.044,Z 668.053,A -85,B 0,C 180,E1 16784.155,E2 16784.155} C_VEL
LIN {X 0,Y 288.319,Z 698.679,A -85,B 0,C 180,E1 16789.918,E2 16789.918} C_VEL
LIN {X 0,Y 276.82,Z 723.914,A -85,B 0,C 180,E1 16796.84,E2 16796.84} C_VEL
LIN {X 0,Y 268.593,Z 743.822,A -85,B 0,C 180,E1 16804.81,E2 16804.81} C_VEL
LIN {X 0,Y 264.228,Z 757.816,A -85,B 0,C 180,E1 16813.35,E2 16813.35} C_VEL
LIN {X 0,Y 262.946,Z 765.725,A -85,B 0,C 180,E1 16821.723,E2 16821.723} C_VEL
LIN {X 0,Y 263.121,Z 768.192,A -85,B 0,C 180,E1 16829.999,E2 16829.999} C_VEL
LIN {X 0,Y 262.923,Z 766.217,A -85,B 0,C 180,E1 16836.613,E2 16836.613} C_VEL
LIN {X 0,Y 263.543,Z 760.649,A -85,B 0,C 180,E1 16843.285,E2 16843.285} C_VEL
LIN {X 0,Y 266.273,Z 748.147,A -85,B 0,C 180,E1 16851.691,E2 16851.691} C_VEL
LIN {X 0,Y 272.285,Z 729.952,A -85,B 0,C 180,E1 16859.571,E2 16859.571} C_VEL
LIN {X 0,Y 281.019,Z 707.2,A -85,B 0,C 180,E1 16866.346,E2 16866.346} C_VEL
LIN {X 0,Y 292.04,Z 678.369,A -85,B 0,C 180,E1 16872.376,E2 16872.376} C_VEL
LIN {X 0,Y 303.541,Z 645.982,A -85,B 0,C 180,E1 16877.107,E2 16877.107} C_VEL
LIN {X 0,Y 314.518,Z 609.778,A -85,B 0,C 180,E1 16880.759,E2 16880.759} C_VEL
LIN {X 0,Y 318.839,Z 593.056,A -85,B 0,C 180,E1 16882.112,E2 16882.112} C_VEL
LIN {X 0,Y 308.707,Z 565.06,A -85,B 0,C 180,E1 16887.262,E2 16887.262} C_VEL
LIN {X 0,Y 303.735,Z 558.242,A -85,B 0,C 180,E1 16889.141,E2 16889.141} C_VEL
LIN {X 0,Y 294.534,Z 548.494,A -85,B 0,C 180,E1 16892.511,E2 16892.511} C_VEL
LIN {X 0,Y 283.144,Z 524.959,A -85,B 0,C 180,E1 16898.848,E2 16898.848} C_VEL
LIN {X 0,Y 273.328,Z 507.561,A -85,B 0,C 180,E1 16905.161,E2 16905.161} C_VEL
LIN {X 0,Y 267.001,Z 496.756,A -85,B 0,C 180,E1 16910.211,E2 16910.211} C_VEL
LIN {X 0,Y 263.058,Z 490.14,A -85,B 0,C 180,E1 16914.224,E2 16914.224} C_VEL
LIN {X 0,Y 259.804,Z 484.2,A -85,B 0,C 180,E1 16918.649,E2 16918.649} C_VEL
LIN {X 0,Y 255.763,Z 481.246,A -85,B 0,C 180,E1 16926.805,E2 16926.805} C_VEL
LIN {X 0,Y 256.924,Z 482.969,A -85,B 0,C 180,E1 16938.028,E2 16938.028} C_VEL
LIN {X 0,Y 258.373,Z 484.661,A -85,B 0,C 180,E1 16940.842,E2 16940.842} C_VEL
LIN {X 0,Y 262.253,Z 490.5,A -85,B 0,C 180,E1 16946.122,E2 16946.122} C_VEL
LIN {X 0,Y 267.751,Z 499.56,A -85,B 0,C 180,E1 16951.447,E2 16951.447} C_VEL
LIN {X 0,Y 276.166,Z 512.692,A -85,B 0,C 180,E1 16957.266,E2 16957.266} C_VEL
LIN {X 0,Y 286.315,Z 530.216,A -85,B 0,C 180,E1 16962.815,E2 16962.815} C_VEL
LIN {X 0,Y 296.291,Z 551.631,A -85,B 0,C 180,E1 16968.176,E2 16968.176} C_VEL
LIN {X 0,Y 303.939,Z 576.942,A -85,B 0,C 180,E1 16973.515,E2 16973.515} C_VEL
LIN {X 0,Y 307.482,Z 596.911,A -85,B 0,C 180,E1 16977.496,E2 16977.496} C_VEL
LIN {X 0,Y 295.872,Z 629.029,A -85,B 0,C 180,E1 16981.748,E2 16981.748} C_VEL
LIN {X 0,Y 283.592,Z 657.757,A -85,B 0,C 180,E1 16987.228,E2 16987.228} C_VEL
LIN {X 0,Y 272.374,Z 681.839,A -85,B 0,C 180,E1 16993.863,E2 16993.863} C_VEL
LIN {X 0,Y 263.398,Z 701.245,A -85,B 0,C 180,E1 17001.738,E2 17001.738} C_VEL
LIN {X 0,Y 258.114,Z 714.473,A -85,B 0,C 180,E1 17010.001,E2 17010.001} C_VEL
LIN {X 0,Y 255.543,Z 722.491,A -85,B 0,C 180,E1 17018.519,E2 17018.519} C_VEL
LIN {X 0,Y 254.402,Z 725.64,A -85,B 0,C 180,E1 17027.313,E2 17027.313} C_VEL
LIN {X 0,Y 255.188,Z 724.391,A -85,B 0,C 180,E1 17034.541,E2 17034.541} C_VEL
LIN {X 0,Y 257.563,Z 719.644,A -85,B 0,C 180,E1 17041.944,E2 17041.944} C_VEL
LIN {X 0,Y 262.899,Z 709.077,A -85,B 0,C 180,E1 17050.64,E2 17050.64} C_VEL
LIN {X 0,Y 271.595,Z 694.037,A -85,B 0,C 180,E1 17058.383,E2 17058.383} C_VEL
LIN {X 0,Y 284.285,Z 672.391,A -85,B 0,C 180,E1 17065.776,E2 17065.776} C_VEL
LIN {X 0,Y 298.397,Z 646.451,A -85,B 0,C 180,E1 17071.707,E2 17071.707} C_VEL
LIN {X 0,Y 300.687,Z 641.983,A -85,B 0,C 180,E1 17072.531,E2 17072.531} C_VEL
LIN {X 0,Y 276.847,Z 646.621,A -85,B 0,C 180,E1 17078.398,E2 17078.398} C_VEL
LIN {X 0,Y 260.579,Z 648.951,A -85,B 0,C 180,E1 17085.269,E2 17085.269} C_VEL
LIN {X 0,Y 259.096,Z 663.755,A -85,B 0,C 180,E1 17090.748,E2 17090.748} C_VEL
LIN {X 0,Y 258.734,Z 674.178,A -85,B 0,C 180,E1 17096.64,E2 17096.64} C_VEL
LIN {X 0,Y 259.341,Z 679.236,A -85,B 0,C 180,E1 17101.668,E2 17101.668} C_VEL
LIN {X 0,Y 260.908,Z 680.954,A -85,B 0,C 180,E1 17106.659,E2 17106.659} C_VEL
LIN {X 0,Y 264.689,Z 678.081,A -85,B 0,C 180,E1 17113.221,E2 17113.221} C_VEL
LIN {X 0,Y 269.861,Z 670.437,A -85,B 0,C 180,E1 17118.815,E2 17118.815} C_VEL
LIN {X 0,Y 277.346,Z 656.22,A -85,B 0,C 180,E1 17124.592,E2 17124.592} C_VEL
LIN {X 0,Y 286.231,Z 635.82,A -85,B 0,C 180,E1 17129.723,E2 17129.723} C_VEL
LIN {X 0,Y 289.312,Z 628.991,A -85,B 0,C 180,E1 17131.11,E2 17131.11} C_VEL
LIN {X 0,Y 307.361,Z 616,A -85,B 0,C 180,E1 17134.144,E2 17134.144} C_VEL
LIN {X 0,Y 320.527,Z 604.211,A -85,B 0,C 180,E1 17135.806,E2 17135.806} C_VEL
LIN {X 0,Y 308.231,Z 640.416,A -85,B 0,C 180,E1 17139.339,E2 17139.339} C_VEL
LIN {X 0,Y 294.633,Z 672.269,A -85,B 0,C 180,E1 17143.724,E2 17143.724} C_VEL
LIN {X 0,Y 280.536,Z 701.773,A -85,B 0,C 180,E1 17149.633,E2 17149.633} C_VEL
LIN {X 0,Y 269.121,Z 725.446,A -85,B 0,C 180,E1 17156.544,E2 17156.544} C_VEL
LIN {X 0,Y 260.619,Z 744.74,A -85,B 0,C 180,E1 17164.778,E2 17164.778} C_VEL
LIN {X 0,Y 256.236,Z 758.305,A -85,B 0,C 180,E1 17173.699,E2 17173.699} C_VEL
LIN {X 0,Y 255.085,Z 765.115,A -85,B 0,C 180,E1 17181.466,E2 17181.466} C_VEL
LIN {X 0,Y 255.261,Z 767.535,A -85,B 0,C 180,E1 17189.999,E2 17189.999} C_VEL
LIN {X 0,Y 255.038,Z 765.507,A -85,B 0,C 180,E1 17196.819,E2 17196.819} C_VEL
LIN {X 0,Y 255.694,Z 759.856,A -85,B 0,C 180,E1 17203.701,E2 17203.701} C_VEL
LIN {X 0,Y 258.683,Z 747.255,A -85,B 0,C 180,E1 17212.361,E2 17212.361} C_VEL
LIN {X 0,Y 265.125,Z 728.91,A -85,B 0,C 180,E1 17220.453,E2 17220.453} C_VEL
LIN {X 0,Y 274.36,Z 705.995,A -85,B 0,C 180,E1 17227.376,E2 17227.376} C_VEL
LIN {X 0,Y 285.894,Z 676.882,A -85,B 0,C 180,E1 17233.51,E2 17233.51} C_VEL
LIN {X 0,Y 298.014,Z 643.872,A -85,B 0,C 180,E1 17238.324,E2 17238.324} C_VEL
LIN {X 0,Y 309.371,Z 607.451,A -85,B 0,C 180,E1 17241.941,E2 17241.941} C_VEL
LIN {X 0,Y 312.171,Z 595.258,A -85,B 0,C 180,E1 17243.011,E2 17243.011} C_VEL
LIN {X 0,Y 299.857,Z 561.145,A -85,B 0,C 180,E1 17249.68,E2 17249.68} C_VEL
LIN {X 0,Y 294.534,Z 548.494,A -85,B 0,C 180,E1 17252.511,E2 17252.511} C_VEL
LIN {X 0,Y 289.536,Z 542.642,A -85,B 0,C 180,E1 17254.601,E2 17254.601} C_VEL
LIN {X 0,Y 281.526,Z 535.725,A -85,B 0,C 180,E1 17257.994,E2 17257.994} C_VEL
LIN {X 0,Y 280.92,Z 534.543,A -85,B 0,C 180,E1 17258.354,E2 17258.354} C_VEL
LIN {X 0,Y 270.914,Z 515.726,A -85,B 0,C 180,E1 17265.026,E2 17265.026} C_VEL
LIN {X 0,Y 263.839,Z 503.536,A -85,B 0,C 180,E1 17270.926,E2 17270.926} C_VEL
LIN {X 0,Y 260.234,Z 497.249,A -85,B 0,C 180,E1 17274.868,E2 17274.868} C_VEL
LIN {X 0,Y 256.896,Z 490.738,A -85,B 0,C 180,E1 17280.005,E2 17280.005} C_VEL
LIN {X 0,Y 253.259,Z 488.798,A -85,B 0,C 180,E1 17291.08,E2 17291.08} C_VEL
LIN {X 0,Y 256.068,Z 491.976,A -85,B 0,C 180,E1 17300.398,E2 17300.398} C_VEL
LIN {X 0,Y 260.115,Z 498.091,A -85,B 0,C 180,E1 17306.057,E2 17306.057} C_VEL
LIN {X 0,Y 265.394,Z 507.554,A -85,B 0,C 180,E1 17311.357,E2 17311.357} C_VEL
LIN {X 0,Y 273.118,Z 519.81,A -85,B 0,C 180,E1 17316.855,E2 17316.855} C_VEL
LIN {X 0,Y 282.975,Z 537.582,A -85,B 0,C 180,E1 17322.571,E2 17322.571} C_VEL
LIN {X 0,Y 292.255,Z 559.374,A -85,B 0,C 180,E1 17328.13,E2 17328.13} C_VEL
LIN {X 0,Y 298.874,Z 584.696,A -85,B 0,C 180,E1 17333.622,E2 17333.622} C_VEL
LIN {X 0,Y 301.07,Z 599.703,A -85,B 0,C 180,E1 17336.715,E2 17336.715} C_VEL
LIN {X 0,Y 289.103,Z 631.376,A -85,B 0,C 180,E1 17341.024,E2 17341.024} C_VEL
LIN {X 0,Y 276.48,Z 659.673,A -85,B 0,C 180,E1 17346.607,E2 17346.607} C_VEL
LIN {X 0,Y 264.916,Z 683.469,A -85,B 0,C 180,E1 17353.396,E2 17353.396} C_VEL
LIN {X 0,Y 255.662,Z 702.578,A -85,B 0,C 180,E1 17361.486,E2 17361.486} C_VEL
LIN {X 0,Y 250.227,Z 715.581,A -85,B 0,C 180,E1 17370.001,E2 17370.001} C_VEL
LIN {X 0,Y 247.586,Z 723.403,A -85,B 0,C 180,E1 17378.795,E2 17378.795} C_VEL
LIN {X 0,Y 246.516,Z 726.345,A -85,B 0,C 180,E1 17387.885,E2 17387.885} C_VEL
LIN {X 0,Y 247.932,Z 724.26,A -85,B 0,C 180,E1 17396.787,E2 17396.787} C_VEL
LIN {X 0,Y 251.834,Z 716.796,A -85,B 0,C 180,E1 17406.08,E2 17406.08} C_VEL
LIN {X 0,Y 259.487,Z 703.635,A -85,B 0,C 180,E1 17415.144,E2 17415.144} C_VEL
LIN {X 0,Y 271.528,Z 684.376,A -85,B 0,C 180,E1 17423.378,E2 17423.378} C_VEL
LIN {X 0,Y 285.866,Z 660.424,A -85,B 0,C 180,E1 17430.134,E2 17430.134} C_VEL
LIN {X 0,Y 292.111,Z 648.538,A -85,B 0,C 180,E1 17432.715,E2 17432.715} C_VEL
LIN {X 0,Y 265.658,Z 653.123,A -85,B 0,C 180,E1 17439.999,E2 17439.999} C_VEL
LIN {X 0,Y 252.215,Z 654.27,A -85,B 0,C 180,E1 17446.544,E2 17446.544} C_VEL
LIN {X 0,Y 250.963,Z 669.566,A -85,B 0,C 180,E1 17453.065,E2 17453.065} C_VEL
LIN {X 0,Y 251.377,Z 679.04,A -85,B 0,C 180,E1 17459.995,E2 17459.995} C_VEL
LIN {X 0,Y 253.219,Z 682.524,A -85,B 0,C 180,E1 17466.863,E2 17466.863} C_VEL
LIN {X 0,Y 257.285,Z 680.119,A -85,B 0,C 180,E1 17473.609,E2 17473.609} C_VEL
LIN {X 0,Y 262.822,Z 672.999,A -85,B 0,C 180,E1 17479.338,E2 17479.338} C_VEL
LIN {X 0,Y 270.821,Z 659.577,A -85,B 0,C 180,E1 17485.226,E2 17485.226} C_VEL
LIN {X 0,Y 280.204,Z 640.423,A -85,B 0,C 180,E1 17490.384,E2 17490.384} C_VEL
LIN {X 0,Y 281.04,Z 638.615,A -85,B 0,C 180,E1 17490.777,E2 17490.777} C_VEL
LIN {X 0,Y 299.845,Z 626.917,A -85,B 0,C 180,E1 17494.17,E2 17494.17} C_VEL
LIN {X 0,Y 312.193,Z 617.31,A -85,B 0,C 180,E1 17495.796,E2 17495.796} C_VEL
LIN {X 0,Y 298.078,Z 652.681,A -85,B 0,C 180,E1 17499.643,E2 17499.643} C_VEL
LIN {X 0,Y 283.416,Z 684.028,A -85,B 0,C 180,E1 17504.699,E2 17504.699} C_VEL
LIN {X 0,Y 269.972,Z 710.374,A -85,B 0,C 180,E1 17510.879,E2 17510.879} C_VEL
LIN {X 0,Y 258.39,Z 733.1,A -85,B 0,C 180,E1 17518.663,E2 17518.663} C_VEL
LIN {X 0,Y 251.227,Z 749.35,A -85,B 0,C 180,E1 17526.936,E2 17526.936} C_VEL
LIN {X 0,Y 247.805,Z 760.516,A -85,B 0,C 180,E1 17535.853,E2 17535.853} C_VEL
LIN {X 0,Y 247.128,Z 765.415,A -85,B 0,C 180,E1 17542.961,E2 17542.961} C_VEL
LIN {X 0,Y 247.38,Z 766.875,A -85,B 0,C 180,E1 17549.999,E2 17549.999} C_VEL
LIN {X 0,Y 247.156,Z 764.793,A -85,B 0,C 180,E1 17557.037,E2 17557.037} C_VEL
LIN {X 0,Y 248.025,Z 758.062,A -85,B 0,C 180,E1 17565.037,E2 17565.037} C_VEL
LIN {X 0,Y 251.657,Z 744.745,A -85,B 0,C 180,E1 17573.961,E2 17573.961} C_VEL
LIN {X 0,Y 258.523,Z 726.689,A -85,B 0,C 180,E1 17581.81,E2 17581.81} C_VEL
LIN {X 0,Y 268.428,Z 703.115,A -85,B 0,C 180,E1 17588.867,E2 17588.867} C_VEL
LIN {X 0,Y 280.704,Z 673.553,A -85,B 0,C 180,E1 17595.005,E2 17595.005} C_VEL
LIN {X 0,Y 292.999,Z 640.69,A -85,B 0,C 180,E1 17599.697,E2 17599.697} C_VEL
LIN {X 0,Y 304.951,Z 603.006,A -85,B 0,C 180,E1 17603.328,E2 17603.328} C_VEL
LIN {X 0,Y 305.543,Z 597.436,A -85,B 0,C 180,E1 17603.96,E2 17603.96} C_VEL
LIN {X 0,Y 293.977,Z 564.382,A -85,B 0,C 180,E1 17610.715,E2 17610.715} C_VEL
LIN {X 0,Y 282.845,Z 538.548,A -85,B 0,C 180,E1 17617.17,E2 17617.17} C_VEL
LIN {X 0,Y 280.92,Z 534.543,A -85,B 0,C 180,E1 17618.354,E2 17618.354} C_VEL
LIN {X 0,Y 276.308,Z 529.688,A -85,B 0,C 180,E1 17620.674,E2 17620.674} C_VEL
LIN {X 0,Y 268.955,Z 524.886,A -85,B 0,C 180,E1 17624.459,E2 17624.459} C_VEL
LIN {X 0,Y 268.416,Z 523.928,A -85,B 0,C 180,E1 17624.871,E2 17624.871} C_VEL
LIN {X 0,Y 260.78,Z 510.364,A -85,B 0,C 180,E1 17631.555,E2 17631.555} C_VEL
LIN {X 0,Y 257.472,Z 504.448,A -85,B 0,C 180,E1 17635.368,E2 17635.368} C_VEL
LIN {X 0,Y 254.476,Z 498.221,A -85,B 0,C 180,E1 17640.431,E2 17640.431} C_VEL
LIN {X 0,Y 251.162,Z 496.433,A -85,B 0,C 180,E1 17651.174,E2 17651.174} C_VEL
LIN {X 0,Y 253.838,Z 499.559,A -85,B 0,C 180,E1 17660.13,E2 17660.13} C_VEL
LIN {X 0,Y 258.391,Z 507.31,A -85,B 0,C 180,E1 17666.713,E2 17666.713} C_VEL
LIN {X 0,Y 262.8,Z 515.108,A -85,B 0,C 180,E1 17671.124,E2 17671.124} C_VEL
LIN {X 0,Y 272.156,Z 530.078,A -85,B 0,C 180,E1 17677.735,E2 17677.735} C_VEL
LIN {X 0,Y 282.812,Z 552.49,A -85,B 0,C 180,E1 17684.472,E2 17684.472} C_VEL
LIN {X 0,Y 289.92,Z 574.34,A -85,B 0,C 180,E1 17689.785,E2 17689.785} C_VEL
LIN {X 0,Y 294.623,Z 599.498,A -85,B 0,C 180,E1 17695.314,E2 17695.314} C_VEL
LIN {X 0,Y 294.09,Z 604.252,A -85,B 0,C 180,E1 17696.102,E2 17696.102} C_VEL
LIN {X 0,Y 281.521,Z 635.579,A -85,B 0,C 180,E1 17700.609,E2 17700.609} C_VEL
LIN {X 0,Y 268.683,Z 663.059,A -85,B 0,C 180,E1 17706.328,E2 17706.328} C_VEL
LIN {X 0,Y 256.878,Z 686.202,A -85,B 0,C 180,E1 17713.301,E2 17713.301} C_VEL
LIN {X 0,Y 247.95,Z 703.886,A -85,B 0,C 180,E1 17721.219,E2 17721.219} C_VEL
LIN {X 0,Y 242.265,Z 716.901,A -85,B 0,C 180,E1 17730.182,E2 17730.182} C_VEL
LIN {X 0,Y 239.606,Z 724.313,A -85,B 0,C 180,E1 17739.09,E2 17739.09} C_VEL
LIN {X 0,Y 238.633,Z 727.024,A -85,B 0,C 180,E1 17748.497,E2 17748.497} C_VEL
LIN {X 0,Y 240.478,Z 724.398,A -85,B 0,C 180,E1 17758.175,E2 17758.175} C_VEL
LIN {X 0,Y 244.575,Z 717.212,A -85,B 0,C 180,E1 17767.08,E2 17767.08} C_VEL
LIN {X 0,Y 252.531,Z 704.541,A -85,B 0,C 180,E1 17776.013,E2 17776.013} C_VEL
LIN {X 0,Y 264.498,Z 686.508,A -85,B 0,C 180,E1 17784.02,E2 17784.02} C_VEL
LIN {X 0,Y 278.94,Z 663.612,A -85,B 0,C 180,E1 17790.753,E2 17790.753} C_VEL
LIN {X 0,Y 283.362,Z 656.185,A -85,B 0,C 180,E1 17792.433,E2 17792.433} C_VEL
LIN {X 0,Y 283.065,Z 655.014,A -85,B 0,C 180,E1 17792.987,E2 17792.987} C_VEL
LIN {X 0,Y 260.244,Z 658.637,A -85,B 0,C 180,E1 17799.565,E2 17799.565} C_VEL
LIN {X 0,Y 243.837,Z 660.438,A -85,B 0,C 180,E1 17808.352,E2 17808.352} C_VEL
LIN {X 0,Y 243.086,Z 674.289,A -85,B 0,C 180,E1 17815.28,E2 17815.28} C_VEL
LIN {X 0,Y 243.747,Z 681.708,A -85,B 0,C 180,E1 17821.774,E2 17821.774} C_VEL
LIN {X 0,Y 245.542,Z 684.099,A -85,B 0,C 180,E1 17827.078,E2 17827.078} C_VEL
LIN {X 0,Y 249.896,Z 682.19,A -85,B 0,C 180,E1 17834.019,E2 17834.019} C_VEL
LIN {X 0,Y 256.825,Z 674.29,A -85,B 0,C 180,E1 17840.709,E2 17840.709} C_VEL
LIN {X 0,Y 265.642,Z 660.771,A -85,B 0,C 180,E1 17846.663,E2 17846.663} C_VEL
LIN {X 0,Y 273.931,Z 647.155,A -85,B 0,C 180,E1 17850.741,E2 17850.741} C_VEL
LIN {X 0,Y 294.132,Z 635.717,A -85,B 0,C 180,E1 17854.481,E2 17854.481} C_VEL
LIN {X 0,Y 302.498,Z 630.09,A -85,B 0,C 180,E1 17855.644,E2 17855.644} C_VEL
LIN {X 0,Y 287.842,Z 663.888,A -85,B 0,C 180,E1 17860.001,E2 17860.001} C_VEL
LIN {X 0,Y 271.973,Z 694.781,A -85,B 0,C 180,E1 17865.799,E2 17865.799} C_VEL
LIN {X 0,Y 258.344,Z 719.771,A -85,B 0,C 180,E1 17872.759,E2 17872.759} C_VEL
LIN {X 0,Y 248.016,Z 739.321,A -85,B 0,C 180,E1 17880.764,E2 17880.764} C_VEL
LIN {X 0,Y 241.69,Z 754.128,A -85,B 0,C 180,E1 17889.974,E2 17889.974} C_VEL
LIN {X 0,Y 239.416,Z 762.804,A -85,B 0,C 180,E1 17899.063,E2 17899.063} C_VEL
LIN {X 0,Y 239.2,Z 765.96,A -85,B 0,C 180,E1 17906.37,E2 17906.37} C_VEL
LIN {X 0,Y 239.509,Z 766.217,A -85,B 0,C 180,E1 17909.999,E2 17909.999} C_VEL
LIN {X 0,Y 239.288,Z 764.077,A -85,B 0,C 180,E1 17917.27,E2 17917.27} C_VEL
LIN {X 0,Y 240.252,Z 757.246,A -85,B 0,C 180,E1 17925.535,E2 17925.535} C_VEL
LIN {X 0,Y 244.205,Z 743.816,A -85,B 0,C 180,E1 17934.74,E2 17934.74} C_VEL
LIN {X 0,Y 251.492,Z 725.597,A -85,B 0,C 180,E1 17942.809,E2 17942.809} C_VEL
LIN {X 0,Y 261.938,Z 702.061,A -85,B 0,C 180,E1 17949.958,E2 17949.958} C_VEL
LIN {X 0,Y 274.794,Z 672.333,A -85,B 0,C 180,E1 17956.171,E2 17956.171} C_VEL
LIN {X 0,Y 287.468,Z 639.489,A -85,B 0,C 180,E1 17960.881,E2 17960.881} C_VEL
LIN {X 0,Y 299.56,Z 601.559,A -85,B 0,C 180,E1 17964.557,E2 17964.557} C_VEL
LIN {X 0,Y 288.598,Z 568.886,A -85,B 0,C 180,E1 17971.467,E2 17971.467} C_VEL
LIN {X 0,Y 278.18,Z 543.656,A -85,B 0,C 180,E1 17978.032,E2 17978.032} C_VEL
LIN {X 0,Y 268.416,Z 523.928,A -85,B 0,C 180,E1 17984.871,E2 17984.871} C_VEL
LIN {X 0,Y 264.495,Z 520.37,A -85,B 0,C 180,E1 17987.437,E2 17987.437} C_VEL
LIN {X 0,Y 257.813,Z 517.38,A -85,B 0,C 180,E1 17992.034,E2 17992.034} C_VEL
LIN {X 0,Y 254.522,Z 511.433,A -85,B 0,C 180,E1 17996.061,E2 17996.061} C_VEL
LIN {X 0,Y 251.974,Z 505.698,A -85,B 0,C 180,E1 18000.866,E2 18000.866} C_VEL
LIN {X 0,Y 249.027,Z 504.054,A -85,B 0,C 180,E1 18011.271,E2 18011.271} C_VEL
LIN {X 0,Y 251.46,Z 507.063,A -85,B 0,C 180,E1 18019.802,E2 18019.802} C_VEL
LIN {X 0,Y 255.812,Z 514.7,A -85,B 0,C 180,E1 18026.36,E2 18026.36} C_VEL
LIN {X 0,Y 262.639,Z 526.286,A -85,B 0,C 180,E1 18032.842,E2 18032.842} C_VEL
LIN {X 0,Y 271.471,Z 542.574,A -85,B 0,C 180,E1 18039.145,E2 18039.145} C_VEL
LIN {X 0,Y 280.209,Z 563.85,A -85,B 0,C 180,E1 18045.376,E2 18045.376} C_VEL
LIN {X 0,Y 286.08,Z 586.877,A -85,B 0,C 180,E1 18050.955,E2 18050.955} C_VEL
LIN {X 0,Y 288.423,Z 605.105,A -85,B 0,C 180,E1 18055.036,E2 18055.036} C_VEL
LIN {X 0,Y 275.747,Z 635.813,A -85,B 0,C 180,E1 18059.476,E2 18059.476} C_VEL
LIN {X 0,Y 262.343,Z 663.415,A -85,B 0,C 180,E1 18065.265,E2 18065.265} C_VEL
LIN {X 0,Y 250.026,Z 686.68,A -85,B 0,C 180,E1 18072.375,E2 18072.375} C_VEL
LIN {X 0,Y 240.222,Z 705.199,A -85,B 0,C 180,E1 18080.934,E2 18080.934} C_VEL
LIN {X 0,Y 234.451,Z 717.787,A -85,B 0,C 180,E1 18090.001,E2 18090.001} C_VEL
LIN {X 0,Y 232.084,Z 724.076,A -85,B 0,C 180,E1 18097.498,E2 18097.498} C_VEL
LIN {X 0,Y 230.765,Z 727.3,A -85,B 0,C 180,E1 18105.216,E2 18105.216} C_VEL
LIN {X 0,Y 231.294,Z 727.065,A -85,B 0,C 180,E1 18113.579,E2 18113.579} C_VEL
LIN {X 0,Y 234.366,Z 722.439,A -85,B 0,C 180,E1 18122.871,E2 18122.871} C_VEL
LIN {X 0,Y 241.073,Z 712.032,A -85,B 0,C 180,E1 18132.735,E2 18132.735} C_VEL
LIN {X 0,Y 251.835,Z 696.613,A -85,B 0,C 180,E1 18141.409,E2 18141.409} C_VEL
LIN {X 0,Y 266.516,Z 675.375,A -85,B 0,C 180,E1 18149.075,E2 18149.075} C_VEL
LIN {X 0,Y 275.508,Z 661.366,A -85,B 0,C 180,E1 18152.717,E2 18152.717} C_VEL
LIN {X 0,Y 247.518,Z 664.703,A -85,B 0,C 180,E1 18162.186,E2 18162.186} C_VEL
LIN {X 0,Y 235.645,Z 665.553,A -85,B 0,C 180,E1 18170.051,E2 18170.051} C_VEL
LIN {X 0,Y 235.287,Z 678.037,A -85,B 0,C 180,E1 18177.228,E2 18177.228} C_VEL
LIN {X 0,Y 236.395,Z 684.202,A -85,B 0,C 180,E1 18183.666,E2 18183.666} C_VEL
LIN {X 0,Y 239.932,Z 685.673,A -85,B 0,C 180,E1 18190.907,E2 18190.907} C_VEL
LIN {X 0,Y 245.84,Z 681.409,A -85,B 0,C 180,E1 18197.929,E2 18197.929} C_VEL
LIN {X 0,Y 254.659,Z 670.984,A -85,B 0,C 180,E1 18204.587,E2 18204.587} C_VEL
LIN {X 0,Y 265.542,Z 655.486,A -85,B 0,C 180,E1 18210.393,E2 18210.393} C_VEL
LIN {X 0,Y 286.653,Z 645.098,A -85,B 0,C 180,E1 18214.59,E2 18214.59} C_VEL
LIN {X 0,Y 293.646,Z 641.017,A -85,B 0,C 180,E1 18215.625,E2 18215.625} C_VEL
LIN {X 0,Y 277.894,Z 673.44,A -85,B 0,C 180,E1 18220.288,E2 18220.288} C_VEL
LIN {X 0,Y 261.487,Z 702.754,A -85,B 0,C 180,E1 18226.558,E2 18226.558} C_VEL
LIN {X 0,Y 248.02,Z 726.002,A -85,B 0,C 180,E1 18234.013,E2 18234.013} C_VEL
LIN {X 0,Y 238.048,Z 744.475,A -85,B 0,C 180,E1 18242.913,E2 18242.913} C_VEL
LIN {X 0,Y 233.341,Z 755.637,A -85,B 0,C 180,E1 18251.067,E2 18251.067} C_VEL
LIN {X 0,Y 231.577,Z 762.226,A -85,B 0,C 180,E1 18258.687,E2 18258.687} C_VEL
LIN {X 0,Y 231.306,Z 765.317,A -85,B 0,C 180,E1 18266.246,E2 18266.246} C_VEL
LIN {X 0,Y 231.626,Z 765.557,A -85,B 0,C 180,E1 18269.999,E2 18269.999} C_VEL
LIN {X 0,Y 231.407,Z 763.356,A -85,B 0,C 180,E1 18277.519,E2 18277.519} C_VEL
LIN {X 0,Y 232.49,Z 756.436,A -85,B 0,C 180,E1 18286.068,E2 18286.068} C_VEL
LIN {X 0,Y 236.8,Z 742.869,A -85,B 0,C 180,E1 18295.568,E2 18295.568} C_VEL
LIN {X 0,Y 245.123,Z 723.27,A -85,B 0,C 180,E1 18304.308,E2 18304.308} C_VEL
LIN {X 0,Y 256.857,Z 698.182,A -85,B 0,C 180,E1 18311.8,E2 18311.8} C_VEL
LIN {X 0,Y 269.702,Z 669.551,A -85,B 0,C 180,E1 18317.658,E2 18317.658} C_VEL
LIN {X 0,Y 282.555,Z 636.895,A -85,B 0,C 180,E1 18322.261,E2 18322.261} C_VEL
LIN {X 0,Y 293.288,Z 604.54,A -85,B 0,C 180,E1 18325.406,E2 18325.406} C_VEL
LIN {X 0,Y 283.434,Z 573.868,A -85,B 0,C 180,E1 18332.14,E2 18332.14} C_VEL
LIN {X 0,Y 274.005,Z 549.912,A -85,B 0,C 180,E1 18338.532,E2 18338.532} C_VEL
LIN {X 0,Y 264.373,Z 529.615,A -85,B 0,C 180,E1 18345.813,E2 18345.813} C_VEL
LIN {X 0,Y 257.813,Z 517.38,A -85,B 0,C 180,E1 18352.034,E2 18352.034} C_VEL
LIN {X 0,Y 253.39,Z 516.071,A -85,B 0,C 180,E1 18355.839,E2 18355.839} C_VEL
LIN {X 0,Y 250.338,Z 515.117,A -85,B 0,C 180,E1 18359.262,E2 18359.262} C_VEL
LIN {X 0,Y 250.148,Z 514.492,A -85,B 0,C 180,E1 18359.741,E2 18359.741} C_VEL
LIN {X 0,Y 247.2,Z 511.64,A -85,B 0,C 180,E1 18367.041,E2 18367.041} C_VEL
LIN {X 0,Y 248.629,Z 513.436,A -85,B 0,C 180,E1 18378.19,E2 18378.19} C_VEL
LIN {X 0,Y 253.241,Z 522.137,A -85,B 0,C 180,E1 18386.051,E2 18386.051} C_VEL
LIN {X 0,Y 259.763,Z 533.648,A -85,B 0,C 180,E1 18392.485,E2 18392.485} C_VEL
LIN {X 0,Y 267.902,Z 549.593,A -85,B 0,C 180,E1 18398.799,E2 18398.799} C_VEL
LIN {X 0,Y 275.627,Z 570.251,A -85,B 0,C 180,E1 18405.032,E2 18405.032} C_VEL
LIN {X 0,Y 280.666,Z 593.148,A -85,B 0,C 180,E1 18410.744,E2 18410.744} C_VEL
LIN {X 0,Y 282.12,Z 607.946,A -85,B 0,C 180,E1 18414.159,E2 18414.159} C_VEL
LIN {X 0,Y 269.125,Z 637.97,A -85,B 0,C 180,E1 18418.641,E2 18418.641} C_VEL
LIN {X 0,Y 255.329,Z 665.263,A -85,B 0,C 180,E1 18424.538,E2 18424.538} C_VEL
LIN {X 0,Y 242.619,Z 688.203,A -85,B 0,C 180,E1 18431.819,E2 18431.819} C_VEL
LIN {X 0,Y 232.493,Z 706.494,A -85,B 0,C 180,E1 18440.63,E2 18440.63} C_VEL
LIN {X 0,Y 226.577,Z 718.879,A -85,B 0,C 180,E1 18450.001,E2 18450.001} C_VEL
LIN {X 0,Y 224.113,Z 724.976,A -85,B 0,C 180,E1 18457.766,E2 18457.766} C_VEL
LIN {X 0,Y 222.787,Z 728.268,A -85,B 0,C 180,E1 18467.916,E2 18467.916} C_VEL
LIN {X 0,Y 224.713,Z 726.334,A -85,B 0,C 180,E1 18478.143,E2 18478.143} C_VEL
LIN {X 0,Y 229.062,Z 719.862,A -85,B 0,C 180,E1 18487.51,E2 18487.51} C_VEL
LIN {X 0,Y 237.562,Z 707.993,A -85,B 0,C 180,E1 18496.93,E2 18496.93} C_VEL
LIN {X 0,Y 250.426,Z 690.862,A -85,B 0,C 180,E1 18505.344,E2 18505.344} C_VEL
LIN {X 0,Y 266.122,Z 668.6,A -85,B 0,C 180,E1 18512.426,E2 18512.426} C_VEL
LIN {X 0,Y 267.133,Z 666.614,A -85,B 0,C 180,E1 18513.032,E2 18513.032} C_VEL
LIN {X 0,Y 241.837,Z 669.94,A -85,B 0,C 180,E1 18521.753,E2 18521.753} C_VEL
LIN {X 0,Y 227.494,Z 671.186,A -85,B 0,C 180,E1 18532.345,E2 18532.345} C_VEL
LIN {X 0,Y 227.902,Z 682.217,A -85,B 0,C 180,E1 18539.994,E2 18539.994} C_VEL
LIN {X 0,Y 230.19,Z 687.178,A -85,B 0,C 180,E1 18547.553,E2 18547.553} C_VEL
LIN {X 0,Y 235.162,Z 686.366,A -85,B 0,C 180,E1 18554.917,E2 18554.917} C_VEL
LIN {X 0,Y 243.009,Z 679.769,A -85,B 0,C 180,E1 18561.945,E2 18561.945} C_VEL
LIN {X 0,Y 253.77,Z 666.946,A -85,B 0,C 180,E1 18568.502,E2 18568.502} C_VEL
LIN {X 0,Y 257.133,Z 663.2,A -85,B 0,C 180,E1 18570.026,E2 18570.026} C_VEL
LIN {X 0,Y 277.075,Z 654.786,A -85,B 0,C 180,E1 18574.335,E2 18574.335} C_VEL
LIN {X 0,Y 284.282,Z 651.114,A -85,B 0,C 180,E1 18575.525,E2 18575.525} C_VEL
LIN {X 0,Y 267.461,Z 682.959,A -85,B 0,C 180,E1 18580.767,E2 18580.767} C_VEL
LIN {X 0,Y 251.2,Z 709.986,A -85,B 0,C 180,E1 18587.43,E2 18587.43} C_VEL
LIN {X 0,Y 237.433,Z 732.361,A -85,B 0,C 180,E1 18595.763,E2 18595.763} C_VEL
LIN {X 0,Y 228.197,Z 749.231,A -85,B 0,C 180,E1 18605.499,E2 18605.499} C_VEL
LIN {X 0,Y 224.396,Z 758.801,A -85,B 0,C 180,E1 18614.341,E2 18614.341} C_VEL
LIN {X 0,Y 223.479,Z 763.57,A -85,B 0,C 180,E1 18622.212,E2 18622.212} C_VEL
LIN {X 0,Y 223.758,Z 764.897,A -85,B 0,C 180,E1 18629.999,E2 18629.999} C_VEL
LIN {X 0,Y 223.547,Z 762.632,A -85,B 0,C 180,E1 18637.785,E2 18637.785} C_VEL
LIN {X 0,Y 224.728,Z 755.603,A -85,B 0,C 180,E1 18646.639,E2 18646.639} C_VEL
LIN {X 0,Y 229.407,Z 741.911,A -85,B 0,C 180,E1 18656.455,E2 18656.455} C_VEL
LIN {X 0,Y 237.742,Z 723.389,A -85,B 0,C 180,E1 18664.972,E2 18664.972} C_VEL
LIN {X 0,Y 249.728,Z 698.946,A -85,B 0,C 180,E1 18672.539,E2 18672.539} C_VEL
LIN {X 0,Y 263.527,Z 669.404,A -85,B 0,C 180,E1 18678.737,E2 18678.737} C_VEL
LIN {X 0,Y 276.819,Z 636.996,A -85,B 0,C 180,E1 18683.375,E2 18683.375} C_VEL
LIN {X 0,Y 286.927,Z 607.028,A -85,B 0,C 180,E1 18686.392,E2 18686.392} C_VEL
LIN {X 0,Y 277.62,Z 576.985,A -85,B 0,C 180,E1 18693.267,E2 18693.267} C_VEL
LIN {X 0,Y 268.786,Z 553.707,A -85,B 0,C 180,E1 18699.823,E2 18699.823} C_VEL
LIN {X 0,Y 260.572,Z 535.792,A -85,B 0,C 180,E1 18706.566,E2 18706.566} C_VEL
LIN {X 0,Y 254.266,Z 523.404,A -85,B 0,C 180,E1 18713.166,E2 18713.166} C_VEL
LIN {X 0,Y 250.148,Z 514.492,A -85,B 0,C 180,E1 18719.741,E2 18719.741} C_VEL
LIN {X 0,Y 249.005,Z 513.672,A -85,B 0,C 180,E1 18721.683,E2 18721.683} C_VEL
LIN {X 0,Y 244.784,Z 519.173,A -85,B 0,C 180,E1 18727.723,E2 18727.723} C_VEL
LIN {X 0,Y 246.624,Z 521.362,A -85,B 0,C 180,E1 18738.771,E2 18738.771} C_VEL
LIN {X 0,Y 250.696,Z 529.737,A -85,B 0,C 180,E1 18745.837,E2 18745.837} C_VEL
LIN {X 0,Y 256.696,Z 540.748,A -85,B 0,C 180,E1 18752.067,E2 18752.067} C_VEL
LIN {X 0,Y 263.914,Z 555.87,A -85,B 0,C 180,E1 18758.239,E2 18758.239} C_VEL
LIN {X 0,Y 270.916,Z 576.492,A -85,B 0,C 180,E1 18764.65,E2 18764.65} C_VEL
LIN {X 0,Y 275.189,Z 599.761,A -85,B 0,C 180,E1 18770.653,E2 18770.653} C_VEL
LIN {X 0,Y 275.929,Z 610.502,A -85,B 0,C 180,E1 18773.225,E2 18773.225} C_VEL
LIN {X 0,Y 261.616,Z 642.043,A -85,B 0,C 180,E1 18778.123,E2 18778.123} C_VEL
LIN {X 0,Y 246.761,Z 669.941,A -85,B 0,C 180,E1 18784.564,E2 18784.564} C_VEL
LIN {X 0,Y 233.968,Z 691.805,A -85,B 0,C 180,E1 18792.098,E2 18792.098} C_VEL
LIN {X 0,Y 223.988,Z 709.287,A -85,B 0,C 180,E1 18801.252,E2 18801.252} C_VEL
LIN {X 0,Y 218.677,Z 719.953,A -85,B 0,C 180,E1 18810.001,E2 18810.001} C_VEL
LIN {X 0,Y 216.113,Z 725.876,A -85,B 0,C 180,E1 18818.056,E2 18818.056} C_VEL
LIN {X 0,Y 214.94,Z 728.751,A -85,B 0,C 180,E1 18826.367,E2 18826.367} C_VEL
LIN {X 0,Y 215.816,Z 728.297,A -85,B 0,C 180,E1 18834.895,E2 18834.895} C_VEL
LIN {X 0,Y 219.114,Z 724.052,A -85,B 0,C 180,E1 18843.976,E2 18843.976} C_VEL
LIN {X 0,Y 226.668,Z 714.066,A -85,B 0,C 180,E1 18854.342,E2 18854.342} C_VEL
LIN {X 0,Y 238.192,Z 699.578,A -85,B 0,C 180,E1 18863.125,E2 18863.125} C_VEL
LIN {X 0,Y 254.306,Z 678.743,A -85,B 0,C 180,E1 18871.148,E2 18871.148} C_VEL
LIN {X 0,Y 258.455,Z 672.237,A -85,B 0,C 180,E1 18873.232,E2 18873.232} C_VEL
LIN {X 0,Y 235.984,Z 674.955,A -85,B 0,C 180,E1 18881.284,E2 18881.284} C_VEL
LIN {X 0,Y 219.55,Z 675.913,A -85,B 0,C 180,E1 18894.553,E2 18894.553} C_VEL
LIN {X 0,Y 220.363,Z 685.083,A -85,B 0,C 180,E1 18901.963,E2 18901.963} C_VEL
LIN {X 0,Y 222.505,Z 688.633,A -85,B 0,C 180,E1 18907.815,E2 18907.815} C_VEL
LIN {X 0,Y 227.797,Z 688.408,A -85,B 0,C 180,E1 18915.411,E2 18915.411} C_VEL
LIN {X 0,Y 236.159,Z 682.538,A -85,B 0,C 180,E1 18922.616,E2 18922.616} C_VEL
LIN {X 0,Y 247.585,Z 670.681,A -85,B 0,C 180,E1 18929.282,E2 18929.282} C_VEL
LIN {X 0,Y 271.021,Z 662.12,A -85,B 0,C 180,E1 18934.737,E2 18934.737} C_VEL
LIN {X 0,Y 274.807,Z 660.387,A -85,B 0,C 180,E1 18935.393,E2 18935.393} C_VEL
LIN {X 0,Y 257.989,Z 689.978,A -85,B 0,C 180,E1 18940.919,E2 18940.919} C_VEL
LIN {X 0,Y 242.271,Z 714.457,A -85,B 0,C 180,E1 18947.633,E2 18947.633} C_VEL
LIN {X 0,Y 228.326,Z 735.801,A -85,B 0,C 180,E1 18956.502,E2 18956.502} C_VEL
LIN {X 0,Y 219.536,Z 751.26,A -85,B 0,C 180,E1 18966.635,E2 18966.635} C_VEL
LIN {X 0,Y 216.205,Z 759.753,A -85,B 0,C 180,E1 18975.811,E2 18975.811} C_VEL
LIN {X 0,Y 215.574,Z 762.957,A -85,B 0,C 180,E1 18981.924,E2 18981.924} C_VEL
LIN {X 0,Y 215.873,Z 764.236,A -85,B 0,C 180,E1 18989.999,E2 18989.999} C_VEL
LIN {X 0,Y 215.669,Z 761.898,A -85,B 0,C 180,E1 18998.071,E2 18998.071} C_VEL
LIN {X 0,Y 216.97,Z 754.773,A -85,B 0,C 180,E1 19007.252,E2 19007.252} C_VEL
LIN {X 0,Y 221.699,Z 741.819,A -85,B 0,C 180,E1 19016.865,E2 19016.865} C_VEL
LIN {X 0,Y 230.442,Z 723.381,A -85,B 0,C 180,E1 19025.719,E2 19025.719} C_VEL
LIN {X 0,Y 242.656,Z 699.641,A -85,B 0,C 180,E1 19033.343,E2 19033.343} C_VEL
LIN {X 0,Y 256.575,Z 671.177,A -85,B 0,C 180,E1 19039.534,E2 19039.534} C_VEL
LIN {X 0,Y 270.972,Z 637.544,A -85,B 0,C 180,E1 19044.472,E2 19044.472} C_VEL
LIN {X 0,Y 280.702,Z 609.804,A -85,B 0,C 180,E1 19047.365,E2 19047.365} C_VEL
LIN {X 0,Y 272.249,Z 581.036,A -85,B 0,C 180,E1 19054.228,E2 19054.228} C_VEL
LIN {X 0,Y 263.694,Z 557.533,A -85,B 0,C 180,E1 19061.163,E2 19061.163} C_VEL
LIN {X 0,Y 255.371,Z 538.548,A -85,B 0,C 180,E1 19068.896,E2 19068.896} C_VEL
LIN {X 0,Y 249.21,Z 526.047,A -85,B 0,C 180,E1 19076.664,E2 19076.664} C_VEL
LIN {X 0,Y 246.893,Z 520.921,A -85,B 0,C 180,E1 19081.455,E2 19081.455} C_VEL
LIN {X 0,Y 244.784,Z 519.173,A -85,B 0,C 180,E1 19087.723,E2 19087.723} C_VEL
LIN {X 0,Y 243.832,Z 521.696,A -85,B 0,C 180,E1 19090.727,E2 19090.727} C_VEL
LIN {X 0,Y 242.899,Z 527.577,A -85,B 0,C 180,E1 19095.186,E2 19095.186} C_VEL
LIN {X 0,Y 243.046,Z 527.79,A -85,B 0,C 180,E1 19095.701,E2 19095.701} C_VEL
LIN {X 0,Y 244.386,Z 530.127,A -85,B 0,C 180,E1 19099.409,E2 19099.409} C_VEL
LIN {X 0,Y 247.944,Z 536.956,A -85,B 0,C 180,E1 19105.432,E2 19105.432} C_VEL
LIN {X 0,Y 253.754,Z 548.192,A -85,B 0,C 180,E1 19111.846,E2 19111.846} C_VEL
LIN {X 0,Y 260.336,Z 563.484,A -85,B 0,C 180,E1 19118.17,E2 19118.17} C_VEL
LIN {X 0,Y 266.271,Z 583.641,A -85,B 0,C 180,E1 19124.558,E2 19124.558} C_VEL
LIN {X 0,Y 269.568,Z 606.871,A -85,B 0,C 180,E1 19130.73,E2 19130.73} C_VEL
LIN {X 0,Y 269.728,Z 613.22,A -85,B 0,C 180,E1 19132.278,E2 19132.278} C_VEL
LIN {X 0,Y 255.088,Z 644.139,A -85,B 0,C 180,E1 19137.206,E2 19137.206} C_VEL
LIN {X 0,Y 239.802,Z 671.674,A -85,B 0,C 180,E1 19143.77,E2 19143.77} C_VEL
LIN {X 0,Y 226.561,Z 693.287,A -85,B 0,C 180,E1 19151.492,E2 19151.492} C_VEL
LIN {X 0,Y 216.235,Z 710.501,A -85,B 0,C 180,E1 19160.936,E2 19160.936} C_VEL
LIN {X 0,Y 210.758,Z 720.977,A -85,B 0,C 180,E1 19170.001,E2 19170.001} C_VEL
LIN {X 0,Y 208.151,Z 726.768,A -85,B 0,C 180,E1 19178.366,E2 19178.366} C_VEL
LIN {X 0,Y 207.028,Z 729.553,A -85,B 0,C 180,E1 19188.046,E2 19188.046} C_VEL
LIN {X 0,Y 208.158,Z 728.867,A -85,B 0,C 180,E1 19195.877,E2 19195.877} C_VEL
LIN {X 0,Y 211.678,Z 724.668,A -85,B 0,C 180,E1 19204.907,E2 19204.907} C_VEL
LIN {X 0,Y 219.738,Z 714.866,A -85,B 0,C 180,E1 19215.388,E2 19215.388} C_VEL
LIN {X 0,Y 233.236,Z 698.939,A -85,B 0,C 180,E1 19225.11,E2 19225.11} C_VEL
LIN {X 0,Y 250.485,Z 677.613,A -85,B 0,C 180,E1 19233.116,E2 19233.116} C_VEL
LIN {X 0,Y 223.848,Z 680.362,A -85,B 0,C 180,E1 19244.297,E2 19244.297} C_VEL
LIN {X 0,Y 211.8,Z 680.964,A -85,B 0,C 180,E1 19257.435,E2 19257.435} C_VEL
LIN {X 0,Y 213.058,Z 687.809,A -85,B 0,C 180,E1 19264.069,E2 19264.069} C_VEL
LIN {X 0,Y 217.299,Z 690.948,A -85,B 0,C 180,E1 19272.059,E2 19272.059} C_VEL
LIN {X 0,Y 224.489,Z 688.571,A -85,B 0,C 180,E1 19279.701,E2 19279.701} C_VEL
LIN {X 0,Y 235.091,Z 680.536,A -85,B 0,C 180,E1 19286.789,E2 19286.789} C_VEL
LIN {X 0,Y 240.249,Z 677.098,A -85,B 0,C 180,E1 19289.229,E2 19289.229} C_VEL
LIN {X 0,Y 265.406,Z 668.886,A -85,B 0,C 180,E1 19295.27,E2 19295.27} C_VEL
LIN {X 0,Y 247.465,Z 697.942,A -85,B 0,C 180,E1 19301.451,E2 19301.451} C_VEL
LIN {X 0,Y 230.979,Z 721.804,A -85,B 0,C 180,E1 19309.04,E2 19309.04} C_VEL
LIN {X 0,Y 217.776,Z 741.053,A -85,B 0,C 180,E1 19318.57,E2 19318.57} C_VEL
LIN {X 0,Y 210.175,Z 754.581,A -85,B 0,C 180,E1 19329.447,E2 19329.447} C_VEL
LIN {X 0,Y 208.042,Z 760.462,A -85,B 0,C 180,E1 19337.388,E2 19337.388} C_VEL
LIN {X 0,Y 207.632,Z 763.381,A -85,B 0,C 180,E1 19345.817,E2 19345.817} C_VEL
LIN {X 0,Y 207.988,Z 763.575,A -85,B 0,C 180,E1 19349.999,E2 19349.999} C_VEL
LIN {X 0,Y 207.782,Z 761.151,A -85,B 0,C 180,E1 19358.379,E2 19358.379} C_VEL
LIN {X 0,Y 209.496,Z 753.148,A -85,B 0,C 180,E1 19368.684,E2 19368.684} C_VEL
LIN {X 0,Y 214.795,Z 739.843,A -85,B 0,C 180,E1 19378.475,E2 19378.475} C_VEL
LIN {X 0,Y 225.021,Z 719.935,A -85,B 0,C 180,E1 19387.837,E2 19387.837} C_VEL
LIN {X 0,Y 238.538,Z 694.793,A -85,B 0,C 180,E1 19395.624,E2 19395.624} C_VEL
LIN {X 0,Y 253.26,Z 665.463,A -85,B 0,C 180,E1 19401.69,E2 19401.69} C_VEL
LIN {X 0,Y 267.419,Z 632.726,A -85,B 0,C 180,E1 19406.257,E2 19406.257} C_VEL
LIN {X 0,Y 274.513,Z 612.66,A -85,B 0,C 180,E1 19408.356,E2 19408.356} C_VEL
LIN {X 0,Y 266.748,Z 584.589,A -85,B 0,C 180,E1 19415.354,E2 19415.354} C_VEL
LIN {X 0,Y 259.085,Z 562.619,A -85,B 0,C 180,E1 19422.139,E2 19422.139} C_VEL
LIN {X 0,Y 251.75,Z 544.933,A -85,B 0,C 180,E1 19429.611,E2 19429.611} C_VEL
LIN {X 0,Y 246.042,Z 532.585,A -85,B 0,C 180,E1 19437.628,E2 19437.628} C_VEL
LIN {X 0,Y 243.542,Z 527.447,A -85,B 0,C 180,E1 19443.57,E2 19443.57} C_VEL
LIN {X 0,Y 242.284,Z 526.666,A -85,B 0,C 180,E1 19450.811,E2 19450.811} C_VEL
LIN {X 0,Y 243.046,Z 527.79,A -85,B 0,C 180,E1 19455.701,E2 19455.701} C_VEL
LIN {X 0,Y 243.315,Z 531.942,A -85,B 0,C 180,E1 19458.617,E2 19458.617} C_VEL
LIN {X 0,Y 243.902,Z 541.412,A -85,B 0,C 180,E1 19463.054,E2 19463.054} C_VEL
LIN {X 0,Y 244.083,Z 541.647,A -85,B 0,C 180,E1 19463.305,E2 19463.305} C_VEL
LIN {X 0,Y 249.26,Z 552.442,A -85,B 0,C 180,E1 19470.08,E2 19470.08} C_VEL
LIN {X 0,Y 255.421,Z 567.578,A -85,B 0,C 180,E1 19476.844,E2 19476.844} C_VEL
LIN {X 0,Y 260.695,Z 586.742,A -85,B 0,C 180,E1 19483.28,E2 19483.28} C_VEL
LIN {X 0,Y 263.438,Z 607.99,A -85,B 0,C 180,E1 19489.248,E2 19489.248} C_VEL
LIN {X 0,Y 263.242,Z 616.64,A -85,B 0,C 180,E1 19491.39,E2 19491.39} C_VEL
LIN {X 0,Y 248.635,Z 646.207,A -85,B 0,C 180,E1 19496.243,E2 19496.243} C_VEL
LIN {X 0,Y 232.881,Z 673.384,A -85,B 0,C 180,E1 19502.928,E2 19502.928} C_VEL
LIN {X 0,Y 219.19,Z 694.772,A -85,B 0,C 180,E1 19510.846,E2 19510.846} C_VEL
LIN {X 0,Y 208.489,Z 711.706,A -85,B 0,C 180,E1 19520.596,E2 19520.596} C_VEL
LIN {X 0,Y 202.855,Z 721.984,A -85,B 0,C 180,E1 19530.001,E2 19530.001} C_VEL
LIN {X 0,Y 199.835,Z 728.198,A -85,B 0,C 180,E1 19539.927,E2 19539.927} C_VEL
LIN {X 0,Y 199.155,Z 730.155,A -85,B 0,C 180,E1 19547.705,E2 19547.705} C_VEL
LIN {X 0,Y 200.553,Z 729.38,A -85,B 0,C 180,E1 19556.936,E2 19556.936} C_VEL
LIN {X 0,Y 204.547,Z 725.04,A -85,B 0,C 180,E1 19566.313,E2 19566.313} C_VEL
LIN {X 0,Y 213.536,Z 714.917,A -85,B 0,C 180,E1 19577.101,E2 19577.101} C_VEL
LIN {X 0,Y 227.158,Z 699.91,A -85,B 0,C 180,E1 19586.396,E2 19586.396} C_VEL
LIN {X 0,Y 241.933,Z 682.616,A -85,B 0,C 180,E1 19593.293,E2 19593.293} C_VEL
LIN {X 0,Y 217.715,Z 685.081,A -85,B 0,C 180,E1 19603.843,E2 19603.843} C_VEL
LIN {X 0,Y 204.485,Z 685.836,A -85,B 0,C 180,E1 19620.888,E2 19620.888} C_VEL
LIN {X 0,Y 207.144,Z 691.478,A -85,B 0,C 180,E1 19628.399,E2 19628.399} C_VEL
LIN {X 0,Y 213.135,Z 692.477,A -85,B 0,C 180,E1 19636.501,E2 19636.501} C_VEL
LIN {X 0,Y 222.58,Z 688.059,A -85,B 0,C 180,E1 19644.081,E2 19644.081} C_VEL
LIN {X 0,Y 228.684,Z 683.866,A -85,B 0,C 180,E1 19647.602,E2 19647.602} C_VEL
LIN {X 0,Y 247.803,Z 679.183,A -85,B 0,C 180,E1 19653.352,E2 19653.352} C_VEL
LIN {X 0,Y 256.009,Z 676.641,A -85,B 0,C 180,E1 19655.137,E2 19655.137} C_VEL
LIN {X 0,Y 251.626,Z 684.165,A -85,B 0,C 180,E1 19656.813,E2 19656.813} C_VEL
LIN {X 0,Y 233.017,Z 710.408,A -85,B 0,C 180,E1 19663.625,E2 19663.625} C_VEL
LIN {X 0,Y 216.939,Z 732.178,A -85,B 0,C 180,E1 19672.514,E2 19672.514} C_VEL
LIN {X 0,Y 206.216,Z 747.629,A -85,B 0,C 180,E1 19682.503,E2 19682.503} C_VEL
LIN {X 0,Y 201.139,Z 757.145,A -85,B 0,C 180,E1 19692.475,E2 19692.475} C_VEL
LIN {X 0,Y 199.782,Z 761.743,A -85,B 0,C 180,E1 19701.281,E2 19701.281} C_VEL
LIN {X 0,Y 200.102,Z 762.914,A -85,B 0,C 180,E1 19709.999,E2 19709.999} C_VEL
LIN {X 0,Y 199.903,Z 760.397,A -85,B 0,C 180,E1 19718.712,E2 19718.712} C_VEL
LIN {X 0,Y 201.232,Z 754.125,A -85,B 0,C 180,E1 19727.515,E2 19727.515} C_VEL
LIN {X 0,Y 206.023,Z 742.199,A -85,B 0,C 180,E1 19737.415,E2 19737.415} C_VEL
LIN {X 0,Y 215.959,Z 723.293,A -85,B 0,C 180,E1 19747.35,E2 19747.35} C_VEL
LIN {X 0,Y 229.055,Z 700.181,A -85,B 0,C 180,E1 19755.283,E2 19755.283} C_VEL
LIN {X 0,Y 244.022,Z 672.153,A -85,B 0,C 180,E1 19761.715,E2 19761.715} C_VEL
LIN {X 0,Y 259.383,Z 639.196,A -85,B 0,C 180,E1 19766.762,E2 19766.762} C_VEL
LIN {X 0,Y 268.483,Z 615.919,A -85,B 0,C 180,E1 19769.273,E2 19769.273} C_VEL
LIN {X 0,Y 261.334,Z 588.121,A -85,B 0,C 180,E1 19776.534,E2 19776.534} C_VEL
LIN {X 0,Y 253.858,Z 565.567,A -85,B 0,C 180,E1 19783.954,E2 19783.954} C_VEL
LIN {X 0,Y 247.358,Z 549.496,A -85,B 0,C 180,E1 19791.39,E2 19791.39} C_VEL
LIN {X 0,Y 242.893,Z 539.02,A -85,B 0,C 180,E1 19798.762,E2 19798.762} C_VEL
LIN {X 0,Y 241.1,Z 534.97,A -85,B 0,C 180,E1 19803.606,E2 19803.606} C_VEL
LIN {X 0,Y 239.894,Z 534.229,A -85,B 0,C 180,E1 19810.92,E2 19810.92} C_VEL
LIN {X 0,Y 241.832,Z 537.327,A -85,B 0,C 180,E1 19818.942,E2 19818.942} C_VEL
LIN {X 0,Y 244.083,Z 541.647,A -85,B 0,C 180,E1 19823.305,E2 19823.305} C_VEL
LIN {X 0,Y 245.353,Z 547.418,A -85,B 0,C 180,E1 19826.021,E2 19826.021} C_VEL
LIN {X 0,Y 246.368,Z 560.494,A -85,B 0,C 180,E1 19830.244,E2 19830.244} C_VEL
LIN {X 0,Y 251.742,Z 575.573,A -85,B 0,C 180,E1 19836.978,E2 19836.978} C_VEL
LIN {X 0,Y 255.994,Z 594.611,A -85,B 0,C 180,E1 19843.461,E2 19843.461} C_VEL
LIN {X 0,Y 257.705,Z 616.468,A -85,B 0,C 180,E1 19849.738,E2 19849.738} C_VEL
LIN {X 0,Y 256.486,Z 620.721,A -85,B 0,C 180,E1 19850.548,E2 19850.548} C_VEL
LIN {X 0,Y 241.232,Z 650.02,A -85,B 0,C 180,E1 19855.606,E2 19855.606} C_VEL
LIN {X 0,Y 225.09,Z 676.443,A -85,B 0,C 180,E1 19862.455,E2 19862.455} C_VEL
LIN {X 0,Y 210.555,Z 698.154,A -85,B 0,C 180,E1 19871.12,E2 19871.12} C_VEL
LIN {X 0,Y 199.936,Z 714.252,A -85,B 0,C 180,E1 19881.289,E2 19881.289} C_VEL
LIN {X 0,Y 194.099,Z 724.711,A -85,B 0,C 180,E1 19892.236,E2 19892.236} C_VEL
LIN {X 0,Y 192.162,Z 728.551,A -85,B 0,C 180,E1 19899.068,E2 19899.068} C_VEL
LIN {X 0,Y 191.286,Z 730.859,A -85,B 0,C 180,E1 19908.459,E2 19908.459} C_VEL
LIN {X 0,Y 192.974,Z 729.887,A -85,B 0,C 180,E1 19918.085,E2 19918.085} C_VEL
LIN {X 0,Y 198.454,Z 724.359,A -85,B 0,C 180,E1 19929.235,E2 19929.235} C_VEL
LIN {X 0,Y 209.352,Z 713.197,A -85,B 0,C 180,E1 19940.346,E2 19940.346} C_VEL
LIN {X 0,Y 225.427,Z 696.389,A -85,B 0,C 180,E1 19949.848,E2 19949.848} C_VEL
LIN {X 0,Y 232.045,Z 689.068,A -85,B 0,C 180,E1 19952.818,E2 19952.818} C_VEL
LIN {X 0,Y 232.787,Z 687.537,A -85,B 0,C 180,E1 19953.63,E2 19953.63} C_VEL
LIN {X 0,Y 206.309,Z 690.102,A -85,B 0,C 180,E1 19967.275,E2 19967.275} C_VEL
LIN {X 0,Y 198.352,Z 691.517,A -85,B 0,C 180,E1 19986.568,E2 19986.568} C_VEL
LIN {X 0,Y 204.96,Z 694.526,A -85,B 0,C 180,E1 19996.184,E2 19996.184} C_VEL
LIN {X 0,Y 215.832,Z 690.769,A -85,B 0,C 180,E1 20004.884,E2 20004.884} C_VEL
LIN {X 0,Y 235.509,Z 686.595,A -85,B 0,C 180,E1 20012.294,E2 20012.294} C_VEL
LIN {X 0,Y 246.911,Z 683.632,A -85,B 0,C 180,E1 20015.034,E2 20015.034} C_VEL
LIN {X 0,Y 227.944,Z 709.607,A -85,B 0,C 180,E1 20021.918,E2 20021.918} C_VEL
LIN {X 0,Y 210.745,Z 731.443,A -85,B 0,C 180,E1 20030.928,E2 20030.928} C_VEL
LIN {X 0,Y 198.985,Z 747.165,A -85,B 0,C 180,E1 20041.414,E2 20041.414} C_VEL
LIN {X 0,Y 193.434,Z 756.606,A -85,B 0,C 180,E1 20051.753,E2 20051.753} C_VEL
LIN {X 0,Y 191.904,Z 761.142,A -85,B 0,C 180,E1 20060.92,E2 20060.92} C_VEL
LIN {X 0,Y 192.215,Z 762.248,A -85,B 0,C 180,E1 20069.999,E2 20069.999} C_VEL
LIN {X 0,Y 192.061,Z 759.639,A -85,B 0,C 180,E1 20079.071,E2 20079.071} C_VEL
LIN {X 0,Y 193.941,Z 752.078,A -85,B 0,C 180,E1 20089.536,E2 20089.536} C_VEL
LIN {X 0,Y 199.6,Z 739.43,A -85,B 0,C 180,E1 20099.695,E2 20099.695} C_VEL
LIN {X 0,Y 210.646,Z 720.162,A -85,B 0,C 180,E1 20109.57,E2 20109.57} C_VEL
LIN {X 0,Y 225.517,Z 695.052,A -85,B 0,C 180,E1 20117.837,E2 20117.837} C_VEL
LIN {X 0,Y 241.122,Z 666.42,A -85,B 0,C 180,E1 20124.022,E2 20124.022} C_VEL
LIN {X 0,Y 256.686,Z 633.028,A -85,B 0,C 180,E1 20128.793,E2 20128.793} C_VEL
LIN {X 0,Y 262.373,Z 619.017,A -85,B 0,C 180,E1 20130.284,E2 20130.284} C_VEL
LIN {X 0,Y 256.22,Z 592.769,A -85,B 0,C 180,E1 20137.419,E2 20137.419} C_VEL
LIN {X 0,Y 250.033,Z 572.514,A -85,B 0,C 180,E1 20144.276,E2 20144.276} C_VEL
LIN {X 0,Y 244.474,Z 557.369,A -85,B 0,C 180,E1 20151.288,E2 20151.288} C_VEL
LIN {X 0,Y 240.224,Z 546.616,A -85,B 0,C 180,E1 20158.748,E2 20158.748} C_VEL
LIN {X 0,Y 238.565,Z 542.48,A -85,B 0,C 180,E1 20163.644,E2 20163.644} C_VEL
LIN {X 0,Y 237.445,Z 541.746,A -85,B 0,C 180,E1 20171.034,E2 20171.034} C_VEL
LIN {X 0,Y 239.245,Z 544.48,A -85,B 0,C 180,E1 20178.452,E2 20178.452} C_VEL
LIN {X 0,Y 243.182,Z 553.036,A -85,B 0,C 180,E1 20185.843,E2 20185.843} C_VEL
LIN {X 0,Y 246.368,Z 560.494,A -85,B 0,C 180,E1 20190.244,E2 20190.244} C_VEL
LIN {X 0,Y 247.315,Z 567.882,A -85,B 0,C 180,E1 20192.752,E2 20192.752} C_VEL
LIN {X 0,Y 247.477,Z 582.314,A -85,B 0,C 180,E1 20196.682,E2 20196.682} C_VEL
LIN {X 0,Y 250.833,Z 600.535,A -85,B 0,C 180,E1 20203.059,E2 20203.059} C_VEL
LIN {X 0,Y 251.688,Z 620.794,A -85,B 0,C 180,E1 20209.108,E2 20209.108} C_VEL
LIN {X 0,Y 235.937,Z 650.205,A -85,B 0,C 180,E1 20214.156,E2 20214.156} C_VEL
LIN {X 0,Y 219.145,Z 676.746,A -85,B 0,C 180,E1 20221.077,E2 20221.077} C_VEL
LIN {X 0,Y 204.538,Z 697.665,A -85,B 0,C 180,E1 20229.414,E2 20229.414} C_VEL
LIN {X 0,Y 193.026,Z 714.095,A -85,B 0,C 180,E1 20239.835,E2 20239.835} C_VEL
LIN {X 0,Y 187.03,Z 723.991,A -85,B 0,C 180,E1 20250.001,E2 20250.001} C_VEL
LIN {X 0,Y 184.167,Z 729.391,A -85,B 0,C 180,E1 20259.465,E2 20259.465} C_VEL
LIN {X 0,Y 183.434,Z 731.565,A -85,B 0,C 180,E1 20269.28,E2 20269.28} C_VEL
LIN {X 0,Y 185.474,Z 730.4,A -85,B 0,C 180,E1 20279.329,E2 20279.329} C_VEL
LIN {X 0,Y 191.706,Z 724.676,A -85,B 0,C 180,E1 20290.902,E2 20290.902} C_VEL
LIN {X 0,Y 203.934,Z 713.046,A -85,B 0,C 180,E1 20302.407,E2 20302.407} C_VEL
LIN {X 0,Y 220.492,Z 696.687,A -85,B 0,C 180,E1 20311.611,E2 20311.611} C_VEL
LIN {X 0,Y 224.723,Z 692.086,A -85,B 0,C 180,E1 20313.578,E2 20313.578} C_VEL
LIN {X 0,Y 199.928,Z 694.494,A -85,B 0,C 180,E1 20326.862,E2 20326.862} C_VEL
LIN {X 0,Y 196.708,Z 696.281,A -85,B 0,C 180,E1 20355.85,E2 20355.85} C_VEL
LIN {X 0,Y 209.921,Z 695.208,A -85,B 0,C 180,E1 20365.634,E2 20365.634} C_VEL
LIN {X 0,Y 234.024,Z 691.044,A -85,B 0,C 180,E1 20374.049,E2 20374.049} C_VEL
LIN {X 0,Y 237.787,Z 690.162,A -85,B 0,C 180,E1 20374.955,E2 20374.955} C_VEL
LIN {X 0,Y 217.917,Z 715.286,A -85,B 0,C 180,E1 20382.417,E2 20382.417} C_VEL
LIN {X 0,Y 200.809,Z 735.544,A -85,B 0,C 180,E1 20392.028,E2 20392.028} C_VEL
LIN {X 0,Y 189.162,Z 750.453,A -85,B 0,C 180,E1 20403.88,E2 20403.88} C_VEL
LIN {X 0,Y 184.603,Z 758.707,A -85,B 0,C 180,E1 20415.755,E2 20415.755} C_VEL
LIN {X 0,Y 183.942,Z 761.449,A -85,B 0,C 180,E1 20425.278,E2 20425.278} C_VEL
LIN {X 0,Y 184.328,Z 761.569,A -85,B 0,C 180,E1 20429.999,E2 20429.999} C_VEL
LIN {X 0,Y 184.22,Z 758.824,A -85,B 0,C 180,E1 20439.569,E2 20439.569} C_VEL
LIN {X 0,Y 186.281,Z 751.211,A -85,B 0,C 180,E1 20450.374,E2 20450.374} C_VEL
LIN {X 0,Y 192.56,Z 738.31,A -85,B 0,C 180,E1 20460.984,E2 20460.984} C_VEL
LIN {X 0,Y 204.399,Z 718.87,A -85,B 0,C 180,E1 20471.103,E2 20471.103} C_VEL
LIN {X 0,Y 219.713,Z 694.208,A -85,B 0,C 180,E1 20479.291,E2 20479.291} C_VEL
LIN {X 0,Y 235.681,Z 666.016,A -85,B 0,C 180,E1 20485.431,E2 20485.431} C_VEL
LIN {X 0,Y 251.363,Z 633.612,A -85,B 0,C 180,E1 20490.103,E2 20490.103} C_VEL
LIN {X 0,Y 256.182,Z 622.324,A -85,B 0,C 180,E1 20491.297,E2 20491.297} C_VEL
LIN {X 0,Y 251.532,Z 598.833,A -85,B 0,C 180,E1 20497.908,E2 20497.908} C_VEL
LIN {X 0,Y 245.642,Z 577.785,A -85,B 0,C 180,E1 20505.277,E2 20505.277} C_VEL
LIN {X 0,Y 240.422,Z 562.462,A -85,B 0,C 180,E1 20512.77,E2 20512.77} C_VEL
LIN {X 0,Y 237.048,Z 552.813,A -85,B 0,C 180,E1 20520.006,E2 20520.006} C_VEL
LIN {X 0,Y 235.903,Z 549.956,A -85,B 0,C 180,E1 20523.685,E2 20523.685} C_VEL
LIN {X 0,Y 234.973,Z 549.269,A -85,B 0,C 180,E1 20531.151,E2 20531.151} C_VEL
LIN {X 0,Y 236.772,Z 552.426,A -85,B 0,C 180,E1 20538.652,E2 20538.652} C_VEL
LIN {X 0,Y 240.521,Z 560.982,A -85,B 0,C 180,E1 20546.15,E2 20546.15} C_VEL
LIN {X 0,Y 246.019,Z 576.703,A -85,B 0,C 180,E1 20554.391,E2 20554.391} C_VEL
LIN {X 0,Y 247.477,Z 582.314,A -85,B 0,C 180,E1 20556.682,E2 20556.682} C_VEL
LIN {X 0,Y 247.475,Z 590.805,A -85,B 0,C 180,E1 20559.001,E2 20559.001} C_VEL
LIN {X 0,Y 245.521,Z 606.379,A -85,B 0,C 180,E1 20562.663,E2 20562.663} C_VEL
LIN {X 0,Y 245.751,Z 623.371,A -85,B 0,C 180,E1 20567.949,E2 20567.949} C_VEL
LIN {X 0,Y 228.621,Z 653.9,A -85,B 0,C 180,E1 20573.413,E2 20573.413} C_VEL
LIN {X 0,Y 211.418,Z 679.745,A -85,B 0,C 180,E1 20580.504,E2 20580.504} C_VEL
LIN {X 0,Y 195.848,Z 700.907,A -85,B 0,C 180,E1 20589.642,E2 20589.642} C_VEL
LIN {X 0,Y 184.432,Z 716.611,A -85,B 0,C 180,E1 20600.551,E2 20600.551} C_VEL
LIN {X 0,Y 178.233,Z 726.589,A -85,B 0,C 180,E1 20612.435,E2 20612.435} C_VEL
LIN {X 0,Y 176.145,Z 730.216,A -85,B 0,C 180,E1 20619.9,E2 20619.9} C_VEL
LIN {X 0,Y 175.594,Z 732.274,A -85,B 0,C 180,E1 20630.177,E2 20630.177} C_VEL
LIN {X 0,Y 178.538,Z 730.568,A -85,B 0,C 180,E1 20641.991,E2 20641.991} C_VEL
LIN {X 0,Y 186.453,Z 723.779,A -85,B 0,C 180,E1 20654.325,E2 20654.325} C_VEL
LIN {X 0,Y 200.981,Z 710.939,A -85,B 0,C 180,E1 20665.967,E2 20665.967} C_VEL
LIN {X 0,Y 215.544,Z 697.207,A -85,B 0,C 180,E1 20673.362,E2 20673.362} C_VEL
LIN {X 0,Y 213.325,Z 696.894,A -85,B 0,C 180,E1 20674.79,E2 20674.79} C_VEL
LIN {X 0,Y 189.457,Z 699.051,A -85,B 0,C 180,E1 20690.796,E2 20690.796} C_VEL
LIN {X 0,Y 192.192,Z 700.579,A -85,B 0,C 180,E1 20718.36,E2 20718.36} C_VEL
LIN {X 0,Y 212.498,Z 698.952,A -85,B 0,C 180,E1 20729.909,E2 20729.909} C_VEL
LIN {X 0,Y 227.874,Z 696.351,A -85,B 0,C 180,E1 20734.675,E2 20734.675} C_VEL
LIN {X 0,Y 223.773,Z 702.078,A -85,B 0,C 180,E1 20736.476,E2 20736.476} C_VEL
LIN {X 0,Y 204.315,Z 724.277,A -85,B 0,C 180,E1 20744.626,E2 20744.626} C_VEL
LIN {X 0,Y 187.96,Z 742.452,A -85,B 0,C 180,E1 20755.674,E2 20755.674} C_VEL
LIN {X 0,Y 179.342,Z 753.563,A -85,B 0,C 180,E1 20767.171,E2 20767.171} C_VEL
LIN {X 0,Y 176.8,Z 758.122,A -85,B 0,C 180,E1 20775.112,E2 20775.112} C_VEL
LIN {X 0,Y 176.04,Z 760.807,A -85,B 0,C 180,E1 20785.065,E2 20785.065} C_VEL
LIN {X 0,Y 176.468,Z 760.884,A -85,B 0,C 180,E1 20789.999,E2 20789.999} C_VEL
LIN {X 0,Y 176.352,Z 758.108,A -85,B 0,C 180,E1 20799.887,E2 20799.887} C_VEL
LIN {X 0,Y 178.646,Z 750.373,A -85,B 0,C 180,E1 20811.234,E2 20811.234} C_VEL
LIN {X 0,Y 185.357,Z 737.616,A -85,B 0,C 180,E1 20822.07,E2 20822.07} C_VEL
LIN {X 0,Y 197.406,Z 718.875,A -85,B 0,C 180,E1 20832.153,E2 20832.153} C_VEL
LIN {X 0,Y 213.67,Z 693.951,A -85,B 0,C 180,E1 20840.666,E2 20840.666} C_VEL
LIN {X 0,Y 230.413,Z 665.589,A -85,B 0,C 180,E1 20846.91,E2 20846.91} C_VEL
LIN {X 0,Y 247.254,Z 631.812,A -85,B 0,C 180,E1 20851.736,E2 20851.736} C_VEL
LIN {X 0,Y 250.171,Z 623.979,A -85,B 0,C 180,E1 20852.751,E2 20852.751} C_VEL
LIN {X 0,Y 245.772,Z 600.102,A -85,B 0,C 180,E1 20859.94,E2 20859.94} C_VEL
LIN {X 0,Y 240.619,Z 580.77,A -85,B 0,C 180,E1 20867.283,E2 20867.283} C_VEL
LIN {X 0,Y 236.012,Z 565.94,A -85,B 0,C 180,E1 20875.406,E2 20875.406} C_VEL
LIN {X 0,Y 233.748,Z 558.668,A -85,B 0,C 180,E1 20881.862,E2 20881.862} C_VEL
LIN {X 0,Y 232.459,Z 556.664,A -85,B 0,C 180,E1 20887.49,E2 20887.49} C_VEL
LIN {X 0,Y 233.004,Z 557.731,A -85,B 0,C 180,E1 20895.071,E2 20895.071} C_VEL
LIN {X 0,Y 235.637,Z 563.868,A -85,B 0,C 180,E1 20902.681,E2 20902.681} C_VEL
LIN {X 0,Y 239.679,Z 575.849,A -85,B 0,C 180,E1 20910.361,E2 20910.361} C_VEL
LIN {X 0,Y 243.174,Z 589.695,A -85,B 0,C 180,E1 20916.652,E2 20916.652} C_VEL
LIN {X 0,Y 245.521,Z 606.379,A -85,B 0,C 180,E1 20922.663,E2 20922.663} C_VEL
LIN {X 0,Y 244.13,Z 615.487,A -85,B 0,C 180,E1 20924.881,E2 20924.881} C_VEL
LIN {X 0,Y 236.372,Z 632.61,A -85,B 0,C 180,E1 20927.798,E2 20927.798} C_VEL
LIN {X 0,Y 219.127,Z 660.914,A -85,B 0,C 180,E1 20933.419,E2 20933.419} C_VEL
LIN {X 0,Y 201.85,Z 685.105,A -85,B 0,C 180,E1 20940.819,E2 20940.819} C_VEL
LIN {X 0,Y 187.095,Z 704.129,A -85,B 0,C 180,E1 20949.884,E2 20949.884} C_VEL
LIN {X 0,Y 175.993,Z 718.674,A -85,B 0,C 180,E1 20961.077,E2 20961.077} C_VEL
LIN {X 0,Y 170.276,Z 727.519,A -85,B 0,C 180,E1 20972.549,E2 20972.549} C_VEL
LIN {X 0,Y 168.124,Z 731.039,A -85,B 0,C 180,E1 20980.378,E2 20980.378} C_VEL
LIN {X 0,Y 167.785,Z 732.971,A -85,B 0,C 180,E1 20991.16,E2 20991.16} C_VEL
LIN {X 0,Y 170.692,Z 731.456,A -85,B 0,C 180,E1 21002.157,E2 21002.157} C_VEL
LIN {X 0,Y 178.493,Z 725.459,A -85,B 0,C 180,E1 21014.459,E2 21014.459} C_VEL
LIN {X 0,Y 192.487,Z 713.911,A -85,B 0,C 180,E1 21026.015,E2 21026.015} C_VEL
LIN {X 0,Y 207.082,Z 700.855,A -85,B 0,C 180,E1 21033.974,E2 21033.974} C_VEL
LIN {X 0,Y 182.801,Z 703.168,A -85,B 0,C 180,E1 21050.458,E2 21050.458} C_VEL
LIN {X 0,Y 186.001,Z 705.01,A -85,B 0,C 180,E1 21078.994,E2 21078.994} C_VEL
LIN {X 0,Y 206.967,Z 703.606,A -85,B 0,C 180,E1 21090.794,E2 21090.794} C_VEL
LIN {X 0,Y 218.133,Z 702.048,A -85,B 0,C 180,E1 21094.425,E2 21094.425} C_VEL
LIN {X 0,Y 216.157,Z 705.26,A -85,B 0,C 180,E1 21095.738,E2 21095.738} C_VEL
LIN {X 0,Y 195.524,Z 727.28,A -85,B 0,C 180,E1 21104.542,E2 21104.542} C_VEL
LIN {X 0,Y 179.936,Z 743.456,A -85,B 0,C 180,E1 21115.388,E2 21115.388} C_VEL
LIN {X 0,Y 171.053,Z 754.146,A -85,B 0,C 180,E1 21127.81,E2 21127.81} C_VEL
LIN {X 0,Y 168.276,Z 759.299,A -85,B 0,C 180,E1 21139.632,E2 21139.632} C_VEL
LIN {X 0,Y 168.603,Z 760.199,A -85,B 0,C 180,E1 21149.999,E2 21149.999} C_VEL
LIN {X 0,Y 168.497,Z 757.337,A -85,B 0,C 180,E1 21160.353,E2 21160.353} C_VEL
LIN {X 0,Y 171.073,Z 749.486,A -85,B 0,C 180,E1 21172.223,E2 21172.223} C_VEL
LIN {X 0,Y 178.438,Z 736.584,A -85,B 0,C 180,E1 21183.472,E2 21183.472} C_VEL
LIN {X 0,Y 192.223,Z 716.453,A -85,B 0,C 180,E1 21194.352,E2 21194.352} C_VEL
LIN {X 0,Y 209.253,Z 691.354,A -85,B 0,C 180,E1 21202.743,E2 21202.743} C_VEL
LIN {X 0,Y 227.171,Z 661.836,A -85,B 0,C 180,E1 21209.013,E2 21209.013} C_VEL
LIN {X 0,Y 243.7,Z 629.241,A -85,B 0,C 180,E1 21213.506,E2 21213.506} C_VEL
LIN {X 0,Y 243.969,Z 624.422,A -85,B 0,C 180,E1 21214.647,E2 21214.647} C_VEL
LIN {X 0,Y 240.076,Z 601.486,A -85,B 0,C 180,E1 21222.101,E2 21222.101} C_VEL
LIN {X 0,Y 236.095,Z 584.944,A -85,B 0,C 180,E1 21228.914,E2 21228.914} C_VEL
LIN {X 0,Y 232.242,Z 571.104,A -85,B 0,C 180,E1 21237.203,E2 21237.203} C_VEL
LIN {X 0,Y 230.499,Z 564.875,A -85,B 0,C 180,E1 21243.772,E2 21243.772} C_VEL
LIN {X 0,Y 229.723,Z 564.207,A -85,B 0,C 180,E1 21251.409,E2 21251.409} C_VEL
LIN {X 0,Y 230.726,Z 566.453,A -85,B 0,C 180,E1 21257.181,E2 21257.181} C_VEL
LIN {X 0,Y 233.39,Z 574.056,A -85,B 0,C 180,E1 21264.737,E2 21264.737} C_VEL
LIN {X 0,Y 236.963,Z 587.168,A -85,B 0,C 180,E1 21272.393,E2 21272.393} C_VEL
LIN {X 0,Y 239.556,Z 603.569,A -85,B 0,C 180,E1 21279.205,E2 21279.205} C_VEL
LIN {X 0,Y 240.032,Z 622.298,A -85,B 0,C 180,E1 21285.571,E2 21285.571} C_VEL
LIN {X 0,Y 239.29,Z 627.322,A -85,B 0,C 180,E1 21286.964,E2 21286.964} C_VEL
LIN {X 0,Y 236.372,Z 632.61,A -85,B 0,C 180,E1 21287.798,E2 21287.798} C_VEL
LIN {X 0,Y 226.476,Z 645.767,A -85,B 0,C 180,E1 21289.307,E2 21289.307} C_VEL
LIN {X 0,Y 216.084,Z 658.12,A -85,B 0,C 180,E1 21291.067,E2 21291.067} C_VEL
LIN {X 0,Y 198.043,Z 682.961,A -85,B 0,C 180,E1 21298.291,E2 21298.291} C_VEL
LIN {X 0,Y 181.287,Z 703.614,A -85,B 0,C 180,E1 21307.925,E2 21307.925} C_VEL
LIN {X 0,Y 168.971,Z 718.851,A -85,B 0,C 180,E1 21319.677,E2 21319.677} C_VEL
LIN {X 0,Y 162.308,Z 728.447,A -85,B 0,C 180,E1 21332.674,E2 21332.674} C_VEL
LIN {X 0,Y 160.11,Z 731.86,A -85,B 0,C 180,E1 21340.903,E2 21340.903} C_VEL
LIN {X 0,Y 159.997,Z 733.62,A -85,B 0,C 180,E1 21352.244,E2 21352.244} C_VEL
LIN {X 0,Y 163.436,Z 731.99,A -85,B 0,C 180,E1 21363.771,E2 21363.771} C_VEL
LIN {X 0,Y 170.949,Z 726.685,A -85,B 0,C 180,E1 21375.12,E2 21375.12} C_VEL
LIN {X 0,Y 185.952,Z 715.285,A -85,B 0,C 180,E1 21387.287,E2 21387.287} C_VEL
LIN {X 0,Y 198.686,Z 704.852,A -85,B 0,C 180,E1 21394.006,E2 21394.006} C_VEL
LIN {X 0,Y 173.15,Z 707.52,A -85,B 0,C 180,E1 21414.976,E2 21414.976} C_VEL
LIN {X 0,Y 179.715,Z 709.2,A -85,B 0,C 180,E1 21439.685,E2 21439.685} C_VEL
LIN {X 0,Y 201.38,Z 708.069,A -85,B 0,C 180,E1 21451.746,E2 21451.746} C_VEL
LIN {X 0,Y 209.322,Z 707.125,A -85,B 0,C 180,E1 21454.382,E2 21454.382} C_VEL
LIN {X 0,Y 188.269,Z 728.589,A -85,B 0,C 180,E1 21463.629,E2 21463.629} C_VEL
LIN {X 0,Y 171.947,Z 744.328,A -85,B 0,C 180,E1 21475.083,E2 21475.083} C_VEL
LIN {X 0,Y 162.862,Z 754.527,A -85,B 0,C 180,E1 21488.354,E2 21488.354} C_VEL
LIN {X 0,Y 160.4,Z 758.677,A -85,B 0,C 180,E1 21499.117,E2 21499.117} C_VEL
LIN {X 0,Y 160.732,Z 759.51,A -85,B 0,C 180,E1 21509.999,E2 21509.999} C_VEL
LIN {X 0,Y 160.632,Z 756.555,A -85,B 0,C 180,E1 21520.865,E2 21520.865} C_VEL
LIN {X 0,Y 163.522,Z 748.687,A -85,B 0,C 180,E1 21533.173,E2 21533.173} C_VEL
LIN {X 0,Y 171.632,Z 735.537,A -85,B 0,C 180,E1 21544.988,E2 21544.988} C_VEL
LIN {X 0,Y 186.403,Z 715.233,A -85,B 0,C 180,E1 21556.128,E2 21556.128} C_VEL
LIN {X 0,Y 204.272,Z 689.91,A -85,B 0,C 180,E1 21564.62,E2 21564.62} C_VEL
LIN {X 0,Y 223.156,Z 659.906,A -85,B 0,C 180,E1 21570.875,E2 21570.875} C_VEL
LIN {X 0,Y 238.458,Z 630.028,A -85,B 0,C 180,E1 21575.065,E2 21575.065} C_VEL
LIN {X 0,Y 235.416,Z 607.355,A -85,B 0,C 180,E1 21582.702,E2 21582.702} C_VEL
LIN {X 0,Y 231.817,Z 589.6,A -85,B 0,C 180,E1 21590.409,E2 21590.409} C_VEL
LIN {X 0,Y 228.86,Z 577.482,A -85,B 0,C 180,E1 21598.11,E2 21598.11} C_VEL
LIN {X 0,Y 227.588,Z 572.271,A -85,B 0,C 180,E1 21603.82,E2 21603.82} C_VEL
LIN {X 0,Y 226.885,Z 571.625,A -85,B 0,C 180,E1 21611.554,E2 21611.554} C_VEL
LIN {X 0,Y 227.814,Z 574.053,A -85,B 0,C 180,E1 21617.47,E2 21617.47} C_VEL
LIN {X 0,Y 230.023,Z 581.992,A -85,B 0,C 180,E1 21625.124,E2 21625.124} C_VEL
LIN {X 0,Y 233.018,Z 595.919,A -85,B 0,C 180,E1 21633.088,E2 21633.088} C_VEL
LIN {X 0,Y 234.618,Z 613.246,A -85,B 0,C 180,E1 21640.196,E2 21640.196} C_VEL
LIN {X 0,Y 234.072,Z 628.284,A -85,B 0,C 180,E1 21645.365,E2 21645.365} C_VEL
LIN {X 0,Y 216.084,Z 658.12,A -85,B 0,C 180,E1 21651.067,E2 21651.067} C_VEL
LIN {X 0,Y 205.419,Z 669.785,A -85,B 0,C 180,E1 21653.158,E2 21653.158} C_VEL
LIN {X 0,Y 194.691,Z 680.523,A -85,B 0,C 180,E1 21655.646,E2 21655.646} C_VEL
LIN {X 0,Y 177.315,Z 701.25,A -85,B 0,C 180,E1 21664.726,E2 21664.726} C_VEL
LIN {X 0,Y 164.162,Z 716.385,A -85,B 0,C 180,E1 21675.609,E2 21675.609} C_VEL
LIN {X 0,Y 156.434,Z 726.23,A -85,B 0,C 180,E1 21687.227,E2 21687.227} C_VEL
LIN {X 0,Y 152.862,Z 731.54,A -85,B 0,C 180,E1 21697.866,E2 21697.866} C_VEL
LIN {X 0,Y 151.743,Z 733.922,A -85,B 0,C 180,E1 21707.419,E2 21707.419} C_VEL
LIN {X 0,Y 153.767,Z 733.8,A -85,B 0,C 180,E1 21719.496,E2 21719.496} C_VEL
LIN {X 0,Y 159.96,Z 730.194,A -85,B 0,C 180,E1 21731.499,E2 21731.499} C_VEL
LIN {X 0,Y 173.3,Z 721.151,A -85,B 0,C 180,E1 21744.597,E2 21744.597} C_VEL
LIN {X 0,Y 189.872,Z 708.885,A -85,B 0,C 180,E1 21754.057,E2 21754.057} C_VEL
LIN {X 0,Y 164.553,Z 712.26,A -85,B 0,C 180,E1 21785.271,E2 21785.271} C_VEL
LIN {X 0,Y 179.313,Z 713.33,A -85,B 0,C 180,E1 21804.963,E2 21804.963} C_VEL
LIN {X 0,Y 199.673,Z 711.971,A -85,B 0,C 180,E1 21814.111,E2 21814.111} C_VEL
LIN {X 0,Y 180.658,Z 730.145,A -85,B 0,C 180,E1 21822.831,E2 21822.831} C_VEL
LIN {X 0,Y 163.95,Z 745.189,A -85,B 0,C 180,E1 21834.745,E2 21834.745} C_VEL
LIN {X 0,Y 155.406,Z 753.88,A -85,B 0,C 180,E1 21847.062,E2 21847.062} C_VEL
LIN {X 0,Y 152.532,Z 758.054,A -85,B 0,C 180,E1 21858.548,E2 21858.548} C_VEL
LIN {X 0,Y 152.863,Z 758.82,A -85,B 0,C 180,E1 21869.999,E2 21869.999} C_VEL
LIN {X 0,Y 152.795,Z 755.767,A -85,B 0,C 180,E1 21881.43,E2 21881.43} C_VEL
LIN {X 0,Y 156.062,Z 747.768,A -85,B 0,C 180,E1 21894.351,E2 21894.351} C_VEL
LIN {X 0,Y 166.327,Z 732.659,A -85,B 0,C 180,E1 21907.912,E2 21907.912} C_VEL
LIN {X 0,Y 181.709,Z 712.665,A -85,B 0,C 180,E1 21918.584,E2 21918.584} C_VEL
LIN {X 0,Y 200.552,Z 687.069,A -85,B 0,C 180,E1 21926.908,E2 21926.908} C_VEL
LIN {X 0,Y 219.912,Z 656.889,A -85,B 0,C 180,E1 21932.967,E2 21932.967} C_VEL
LIN {X 0,Y 232.602,Z 633.146,A -85,B 0,C 180,E1 21936.232,E2 21936.232} C_VEL
LIN {X 0,Y 230.405,Z 611.899,A -85,B 0,C 180,E1 21943.789,E2 21943.789} C_VEL
LIN {X 0,Y 227.683,Z 595.415,A -85,B 0,C 180,E1 21951.3,E2 21951.3} C_VEL
LIN {X 0,Y 225.4,Z 583.84,A -85,B 0,C 180,E1 21959.044,E2 21959.044} C_VEL
LIN {X 0,Y 224.554,Z 579.588,A -85,B 0,C 180,E1 21963.872,E2 21963.872} C_VEL
LIN {X 0,Y 223.843,Z 578.983,A -85,B 0,C 180,E1 21971.713,E2 21971.713} C_VEL
LIN {X 0,Y 224.575,Z 581.497,A -85,B 0,C 180,E1 21977.669,E2 21977.669} C_VEL
LIN {X 0,Y 226.221,Z 588.758,A -85,B 0,C 180,E1 21984.733,E2 21984.733} C_VEL
LIN {X 0,Y 228.303,Z 600.97,A -85,B 0,C 180,E1 21992.048,E2 21992.048} C_VEL
LIN {X 0,Y 229.201,Z 617.801,A -85,B 0,C 180,E1 21999.319,E2 21999.319} C_VEL
LIN {X 0,Y 227.919,Z 632.201,A -85,B 0,C 180,E1 22004.398,E2 22004.398} C_VEL
LIN {X 0,Y 209.226,Z 661.241,A -85,B 0,C 180,E1 22010.04,E2 22010.04} C_VEL
LIN {X 0,Y 194.691,Z 680.523,A -85,B 0,C 180,E1 22015.646,E2 22015.646} C_VEL
LIN {X 0,Y 183.866,Z 690.502,A -85,B 0,C 180,E1 22018.539,E2 22018.539} C_VEL
LIN {X 0,Y 173.03,Z 699.52,A -85,B 0,C 180,E1 22021.895,E2 22021.895} C_VEL
LIN {X 0,Y 158.089,Z 715.904,A -85,B 0,C 180,E1 22033.303,E2 22033.303} C_VEL
LIN {X 0,Y 148.54,Z 727.206,A -85,B 0,C 180,E1 22047.08,E2 22047.08} C_VEL
LIN {X 0,Y 145.434,Z 731.549,A -85,B 0,C 180,E1 22055.977,E2 22055.977} C_VEL
LIN {X 0,Y 143.864,Z 734.675,A -85,B 0,C 180,E1 22068.683,E2 22068.683} C_VEL
LIN {X 0,Y 146.376,Z 734.393,A -85,B 0,C 180,E1 22081.146,E2 22081.146} C_VEL
LIN {X 0,Y 153.463,Z 730.609,A -85,B 0,C 180,E1 22093.682,E2 22093.682} C_VEL
LIN {X 0,Y 168.838,Z 720.928,A -85,B 0,C 180,E1 22107.441,E2 22107.441} C_VEL
LIN {X 0,Y 180.805,Z 712.638,A -85,B 0,C 180,E1 22114.149,E2 22114.149} C_VEL
LIN {X 0,Y 162.375,Z 716.749,A -85,B 0,C 180,E1 22156.235,E2 22156.235} C_VEL
LIN {X 0,Y 180.834,Z 717.024,A -85,B 0,C 180,E1 22170.147,E2 22170.147} C_VEL
LIN {X 0,Y 190.062,Z 716.486,A -85,B 0,C 180,E1 22173.882,E2 22173.882} C_VEL
LIN {X 0,Y 181.861,Z 724.255,A -85,B 0,C 180,E1 22177.725,E2 22177.725} C_VEL
LIN {X 0,Y 161.959,Z 740.912,A -85,B 0,C 180,E1 22189.123,E2 22189.123} C_VEL
LIN {X 0,Y 149.486,Z 751.814,A -85,B 0,C 180,E1 22202.883,E2 22202.883} C_VEL
LIN {X 0,Y 144.677,Z 757.43,A -85,B 0,C 180,E1 22217.917,E2 22217.917} C_VEL
LIN {X 0,Y 144.967,Z 758.128,A -85,B 0,C 180,E1 22229.999,E2 22229.999} C_VEL
LIN {X 0,Y 144.951,Z 754.978,A -85,B 0,C 180,E1 22242.058,E2 22242.058} C_VEL
LIN {X 0,Y 148.675,Z 746.846,A -85,B 0,C 180,E1 22255.646,E2 22255.646} C_VEL
LIN {X 0,Y 159.892,Z 731.588,A -85,B 0,C 180,E1 22269.731,E2 22269.731} C_VEL
LIN {X 0,Y 176.305,Z 711.385,A -85,B 0,C 180,E1 22280.616,E2 22280.616} C_VEL
LIN {X 0,Y 196.033,Z 685.632,A -85,B 0,C 180,E1 22288.923,E2 22288.923} C_VEL
LIN {X 0,Y 215.538,Z 656.258,A -85,B 0,C 180,E1 22294.747,E2 22294.747} C_VEL
LIN {X 0,Y 226.876,Z 635.715,A -85,B 0,C 180,E1 22297.672,E2 22297.672} C_VEL
LIN {X 0,Y 225.254,Z 615.208,A -85,B 0,C 180,E1 22305.407,E2 22305.407} C_VEL
LIN {X 0,Y 223.448,Z 601.14,A -85,B 0,C 180,E1 22312.218,E2 22312.218} C_VEL
LIN {X 0,Y 221.842,Z 590.178,A -85,B 0,C 180,E1 22320.006,E2 22320.006} C_VEL
LIN {X 0,Y 221.312,Z 586.854,A -85,B 0,C 180,E1 22323.929,E2 22323.929} C_VEL
LIN {X 0,Y 220.502,Z 586.216,A -85,B 0,C 180,E1 22331.893,E2 22331.893} C_VEL
LIN {X 0,Y 221.1,Z 588.875,A -85,B 0,C 180,E1 22337.9,E2 22337.9} C_VEL
LIN {X 0,Y 222.372,Z 596.523,A -85,B 0,C 180,E1 22345.069,E2 22345.069} C_VEL
LIN {X 0,Y 223.647,Z 607.613,A -85,B 0,C 180,E1 22351.816,E2 22351.816} C_VEL
LIN {X 0,Y 223.741,Z 623.999,A -85,B 0,C 180,E1 22359.063,E2 22359.063} C_VEL
LIN {X 0,Y 222.619,Z 634.056,A -85,B 0,C 180,E1 22362.859,E2 22362.859} C_VEL
LIN {X 0,Y 203.346,Z 663.048,A -85,B 0,C 180,E1 22368.637,E2 22368.637} C_VEL
LIN {X 0,Y 182.873,Z 688.499,A -85,B 0,C 180,E1 22376.735,E2 22376.735} C_VEL
LIN {X 0,Y 173.03,Z 699.52,A -85,B 0,C 180,E1 22381.895,E2 22381.895} C_VEL
LIN {X 0,Y 162.579,Z 707.695,A -85,B 0,C 180,E1 22385.831,E2 22385.831} C_VEL
LIN {X 0,Y 152.687,Z 714.826,A -85,B 0,C 180,E1 22390.417,E2 22390.417} C_VEL
LIN {X 0,Y 142.124,Z 726.392,A -85,B 0,C 180,E1 22403.885,E2 22403.885} C_VEL
LIN {X 0,Y 137.249,Z 732.586,A -85,B 0,C 180,E1 22416.8,E2 22416.8} C_VEL
LIN {X 0,Y 136.012,Z 735.36,A -85,B 0,C 180,E1 22429.511,E2 22429.511} C_VEL
LIN {X 0,Y 139.119,Z 734.997,A -85,B 0,C 180,E1 22442.97,E2 22442.97} C_VEL
LIN {X 0,Y 147.203,Z 731.04,A -85,B 0,C 180,E1 22456.057,E2 22456.057} C_VEL
LIN {X 0,Y 164.195,Z 721.075,A -85,B 0,C 180,E1 22470.074,E2 22470.074} C_VEL
LIN {X 0,Y 172.17,Z 715.888,A -85,B 0,C 180,E1 22474.607,E2 22474.607} C_VEL
LIN {X 0,Y 152.216,Z 719.958,A -85,B 0,C 180,E1 22511.465,E2 22511.465} C_VEL
LIN {X 0,Y 166.875,Z 720.95,A -85,B 0,C 180,E1 22526.968,E2 22526.968} C_VEL
LIN {X 0,Y 180.723,Z 720.57,A -85,B 0,C 180,E1 22533.698,E2 22533.698} C_VEL
LIN {X 0,Y 160.649,Z 736.785,A -85,B 0,C 180,E1 22543.836,E2 22543.836} C_VEL
LIN {X 0,Y 144.275,Z 749.577,A -85,B 0,C 180,E1 22558.348,E2 22558.348} C_VEL
LIN {X 0,Y 138.16,Z 755.261,A -85,B 0,C 180,E1 22570.804,E2 22570.804} C_VEL
LIN {X 0,Y 136.592,Z 757.608,A -85,B 0,C 180,E1 22585.871,E2 22585.871} C_VEL
LIN {X 0,Y 137.094,Z 757.437,A -85,B 0,C 180,E1 22589.999,E2 22589.999} C_VEL
LIN {X 0,Y 137.148,Z 754.194,A -85,B 0,C 180,E1 22602.755,E2 22602.755} C_VEL
LIN {X 0,Y 141.342,Z 745.919,A -85,B 0,C 180,E1 22617.082,E2 22617.082} C_VEL
LIN {X 0,Y 152.02,Z 732.372,A -85,B 0,C 180,E1 22630.344,E2 22630.344} C_VEL
LIN {X 0,Y 168.875,Z 712.816,A -85,B 0,C 180,E1 22641.605,E2 22641.605} C_VEL
LIN {X 0,Y 189.609,Z 687.236,A -85,B 0,C 180,E1 22650.274,E2 22650.274} C_VEL
LIN {X 0,Y 210.661,Z 656.91,A -85,B 0,C 180,E1 22656.403,E2 22656.403} C_VEL
LIN {X 0,Y 221.142,Z 638.927,A -85,B 0,C 180,E1 22658.941,E2 22658.941} C_VEL
LIN {X 0,Y 220.347,Z 619.721,A -85,B 0,C 180,E1 22666.597,E2 22666.597} C_VEL
LIN {X 0,Y 218.993,Z 605.389,A -85,B 0,C 180,E1 22674.054,E2 22674.054} C_VEL
LIN {X 0,Y 218.199,Z 597.429,A -85,B 0,C 180,E1 22680.006,E2 22680.006} C_VEL
LIN {X 0,Y 217.81,Z 593.989,A -85,B 0,C 180,E1 22683.992,E2 22683.992} C_VEL
LIN {X 0,Y 216.966,Z 593.455,A -85,B 0,C 180,E1 22692.315,E2 22692.315} C_VEL
LIN {X 0,Y 217.438,Z 596.264,A -85,B 0,C 180,E1 22698.267,E2 22698.267} C_VEL
LIN {X 0,Y 218.12,Z 602.931,A -85,B 0,C 180,E1 22704.619,E2 22704.619} C_VEL
LIN {X 0,Y 218.857,Z 614.989,A -85,B 0,C 180,E1 22712.017,E2 22712.017} C_VEL
LIN {X 0,Y 218.095,Z 629.681,A -85,B 0,C 180,E1 22718.674,E2 22718.674} C_VEL
LIN {X 0,Y 216.539,Z 637.845,A -85,B 0,C 180,E1 22721.716,E2 22721.716} C_VEL
LIN {X 0,Y 196.337,Z 666.427,A -85,B 0,C 180,E1 22727.564,E2 22727.564} C_VEL
LIN {X 0,Y 175.34,Z 691.209,A -85,B 0,C 180,E1 22735.856,E2 22735.856} C_VEL
LIN {X 0,Y 156.459,Z 710.964,A -85,B 0,C 180,E1 22747.227,E2 22747.227} C_VEL
LIN {X 0,Y 152.687,Z 714.826,A -85,B 0,C 180,E1 22750.417,E2 22750.417} C_VEL
LIN {X 0,Y 143.531,Z 721.073,A -85,B 0,C 180,E1 22755.686,E2 22755.686} C_VEL
LIN {X 0,Y 135.25,Z 726.254,A -85,B 0,C 180,E1 22761.71,E2 22761.71} C_VEL
LIN {X 0,Y 130.344,Z 732.113,A -85,B 0,C 180,E1 22773.296,E2 22773.296} C_VEL
LIN {X 0,Y 128.097,Z 735.941,A -85,B 0,C 180,E1 22788.965,E2 22788.965} C_VEL
LIN {X 0,Y 131.998,Z 735.553,A -85,B 0,C 180,E1 22804.999,E2 22804.999} C_VEL
LIN {X 0,Y 143.036,Z 730.488,A -85,B 0,C 180,E1 22820.561,E2 22820.561} C_VEL
LIN {X 0,Y 161.032,Z 720.613,A -85,B 0,C 180,E1 22833.464,E2 22833.464} C_VEL
LIN {X 0,Y 162.638,Z 719.263,A -85,B 0,C 180,E1 22835.225,E2 22835.225} C_VEL
LIN {X 0,Y 148.857,Z 723.783,A -85,B 0,C 180,E1 22877.756,E2 22877.756} C_VEL
LIN {X 0,Y 170.886,Z 724.4,A -85,B 0,C 180,E1 22893.366,E2 22893.366} C_VEL
LIN {X 0,Y 165.325,Z 729.106,A -85,B 0,C 180,E1 22896.39,E2 22896.39} C_VEL
LIN {X 0,Y 144.591,Z 743.88,A -85,B 0,C 180,E1 22909.118,E2 22909.118} C_VEL
LIN {X 0,Y 133.276,Z 752.288,A -85,B 0,C 180,E1 22922.97,E2 22922.97} C_VEL
LIN {X 0,Y 129.035,Z 756.198,A -85,B 0,C 180,E1 22936.426,E2 22936.426} C_VEL
